LIN {X 0,Y 474.9,Z 291.328,A -85,B 0,C 180,E1 -7380,E2 -7380} C_VEL
LIN {X 0,Y 474.884,Z 291.326,A -85,B 0,C 180,E1 -7382.545,E2 -7382.545} C_VEL
LIN {X 0,Y 474.749,Z 291.35,A -85,B 0,C 180,E1 -7385.948,E2 -7385.948} C_VEL
LIN {X 0,Y 474.718,Z 291.348,A -85,B 0,C 180,E1 -7388.514,E2 -7388.514} C_VEL
LIN {X 0,Y 474.695,Z 291.358,A -85,B 0,C 180,E1 -7391.963,E2 -7391.963} C_VEL
LIN {X 0,Y 474.692,Z 291.354,A -85,B 0,C 180,E1 -7395.777,E2 -7395.777} C_VEL
LIN {X 0,Y 474.655,Z 291.355,A -85,B 0,C 180,E1 -7399.011,E2 -7399.011} C_VEL
LIN {X 0,Y 474.579,Z 291.366,A -85,B 0,C 180,E1 -7401.73,E2 -7401.73} C_VEL
LIN {X 0,Y 474.628,Z 291.364,A -85,B 0,C 180,E1 -7404.495,E2 -7404.495} C_VEL
LIN {X 0,Y 474.665,Z 291.353,A -85,B 0,C 180,E1 -7407.333,E2 -7407.333} C_VEL
LIN {X 0,Y 474.597,Z 291.367,A -85,B 0,C 180,E1 -7410.231,E2 -7410.231} C_VEL
LIN {X 0,Y 474.635,Z 291.358,A -85,B 0,C 180,E1 -7413.221,E2 -7413.221} C_VEL
LIN {X 0,Y 474.581,Z 291.368,A -85,B 0,C 180,E1 -7416.324,E2 -7416.324} C_VEL
LIN {X 0,Y 474.615,Z 291.36,A -85,B 0,C 180,E1 -7419.549,E2 -7419.549} C_VEL
LIN {X 0,Y 474.595,Z 291.369,A -85,B 0,C 180,E1 -7422.937,E2 -7422.937} C_VEL
LIN {X 0,Y 474.597,Z 291.362,A -85,B 0,C 180,E1 -7425.895,E2 -7425.895} C_VEL
LIN {X 0,Y 474.6,Z 291.37,A -85,B 0,C 180,E1 -7429.045,E2 -7429.045} C_VEL
LIN {X 0,Y 474.602,Z 291.362,A -85,B 0,C 180,E1 -7431.706,E2 -7431.706} C_VEL
LIN {X 0,Y 474.617,Z 291.362,A -85,B 0,C 180,E1 -7434.726,E2 -7434.726} C_VEL
LIN {X 0,Y 474.63,Z 291.359,A -85,B 0,C 180,E1 -7437.789,E2 -7437.789} C_VEL
LIN {X 0,Y 474.596,Z 291.365,A -85,B 0,C 180,E1 -7440.891,E2 -7440.891} C_VEL
LIN {X 0,Y 474.578,Z 291.369,A -85,B 0,C 180,E1 -7443.625,E2 -7443.625} C_VEL
LIN {X 0,Y 474.633,Z 291.357,A -85,B 0,C 180,E1 -7446.643,E2 -7446.643} C_VEL
LIN {X 0,Y 474.651,Z 291.357,A -85,B 0,C 180,E1 -7450.09,E2 -7450.09} C_VEL
LIN {X 0,Y 474.643,Z 291.361,A -85,B 0,C 180,E1 -7451.657,E2 -7451.657} C_VEL
LIN {X 0,Y 473.971,Z 291.444,A -85,B 0,C 180,E1 -7452.366,E2 -7452.366} C_VEL
LIN {X 0,Y 471.123,Z 291.802,A -85,B 0,C 180,E1 -7453.518,E2 -7453.518} C_VEL
LIN {X 0,Y 468.714,Z 292.1,A -85,B 0,C 180,E1 -7454.446,E2 -7454.446} C_VEL
LIN {X 0,Y 467.674,Z 292.226,A -85,B 0,C 180,E1 -7455.163,E2 -7455.163} C_VEL
LIN {X 0,Y 467.585,Z 292.237,A -85,B 0,C 180,E1 -7455.406,E2 -7455.406} C_VEL
LIN {X 0,Y 467.636,Z 292.236,A -85,B 0,C 180,E1 -7457.855,E2 -7457.855} C_VEL
LIN {X 0,Y 467.629,Z 292.236,A -85,B 0,C 180,E1 -7461.357,E2 -7461.357} C_VEL
LIN {X 0,Y 467.684,Z 292.306,A -85,B 0,C 180,E1 -7463.313,E2 -7463.313} C_VEL
LIN {X 0,Y 468.568,Z 298.536,A -85,B 0,C 180,E1 -7464.622,E2 -7464.622} C_VEL
LIN {X 0,Y 468.317,Z 310.915,A -85,B 0,C 180,E1 -7467.097,E2 -7467.097} C_VEL
LIN {X 0,Y 471.304,Z 325.673,A -85,B 0,C 180,E1 -7467.437,E2 -7467.437} C_VEL
LIN {X 0,Y 470.534,Z 418.4,A -85,B 0,C 180,E1 -7468.877,E2 -7468.877} C_VEL
LIN {X 0,Y 470.235,Z 431.426,A -85,B 0,C 180,E1 -7469.251,E2 -7469.251} C_VEL
LIN {X 0,Y 469.902,Z 443.958,A -85,B 0,C 180,E1 -7469.786,E2 -7469.786} C_VEL
LIN {X 0,Y 469.513,Z 455.149,A -85,B 0,C 180,E1 -7470.429,E2 -7470.429} C_VEL
LIN {X 0,Y 468.998,Z 466.713,A -85,B 0,C 180,E1 -7471.289,E2 -7471.289} C_VEL
LIN {X 0,Y 468.477,Z 477.124,A -85,B 0,C 180,E1 -7472.257,E2 -7472.257} C_VEL
LIN {X 0,Y 468.064,Z 485.641,A -85,B 0,C 180,E1 -7473.228,E2 -7473.228} C_VEL
LIN {X 0,Y 467.676,Z 493.506,A -85,B 0,C 180,E1 -7474.31,E2 -7474.31} C_VEL
LIN {X 0,Y 467.319,Z 501.212,A -85,B 0,C 180,E1 -7475.61,E2 -7475.61} C_VEL
LIN {X 0,Y 467.128,Z 507.386,A -85,B 0,C 180,E1 -7476.913,E2 -7476.913} C_VEL
LIN {X 0,Y 466.91,Z 512.316,A -85,B 0,C 180,E1 -7478.222,E2 -7478.222} C_VEL
LIN {X 0,Y 466.766,Z 516.123,A -85,B 0,C 180,E1 -7479.534,E2 -7479.534} C_VEL
LIN {X 0,Y 466.713,Z 518.087,A -85,B 0,C 180,E1 -7480.411,E2 -7480.411} C_VEL
LIN {X 0,Y 466.654,Z 520.275,A -85,B 0,C 180,E1 -7481.782,E2 -7481.782} C_VEL
LIN {X 0,Y 466.566,Z 521.392,A -85,B 0,C 180,E1 -7483.059,E2 -7483.059} C_VEL
LIN {X 0,Y 466.536,Z 521.677,A -85,B 0,C 180,E1 -7483.948,E2 -7483.948} C_VEL
LIN {X 0,Y 466.586,Z 521.216,A -85,B 0,C 180,E1 -7485.418,E2 -7485.418} C_VEL
LIN {X 0,Y 466.553,Z 519.949,A -85,B 0,C 180,E1 -7486.632,E2 -7486.632} C_VEL
LIN {X 0,Y 466.652,Z 518.526,A -85,B 0,C 180,E1 -7487.531,E2 -7487.531} C_VEL
LIN {X 0,Y 466.799,Z 515.6,A -85,B 0,C 180,E1 -7488.842,E2 -7488.842} C_VEL
LIN {X 0,Y 466.982,Z 511.277,A -85,B 0,C 180,E1 -7490.252,E2 -7490.252} C_VEL
LIN {X 0,Y 467.214,Z 505.761,A -85,B 0,C 180,E1 -7491.626,E2 -7491.626} C_VEL
LIN {X 0,Y 467.533,Z 498.734,A -85,B 0,C 180,E1 -7493.007,E2 -7493.007} C_VEL
LIN {X 0,Y 467.895,Z 491.468,A -85,B 0,C 180,E1 -7494.162,E2 -7494.162} C_VEL
LIN {X 0,Y 468.379,Z 482.6,A -85,B 0,C 180,E1 -7495.318,E2 -7495.318} C_VEL
LIN {X 0,Y 468.801,Z 473.035,A -85,B 0,C 180,E1 -7496.331,E2 -7496.331} C_VEL
LIN {X 0,Y 469.269,Z 463.203,A -85,B 0,C 180,E1 -7497.18,E2 -7497.18} C_VEL
LIN {X 0,Y 469.812,Z 452.16,A -85,B 0,C 180,E1 -7497.943,E2 -7497.943} C_VEL
LIN {X 0,Y 470.175,Z 440.391,A -85,B 0,C 180,E1 -7498.576,E2 -7498.576} C_VEL
LIN {X 0,Y 470.52,Z 427.541,A -85,B 0,C 180,E1 -7499.072,E2 -7499.072} C_VEL
LIN {X 0,Y 470.719,Z 414.32,A -85,B 0,C 180,E1 -7499.396,E2 -7499.396} C_VEL
LIN {X 0,Y 471.527,Z 325.723,A -85,B 0,C 180,E1 -7500.767,E2 -7500.767} C_VEL
LIN {X 0,Y 468.488,Z 310.771,A -85,B 0,C 180,E1 -7501.149,E2 -7501.149} C_VEL
LIN {X 0,Y 468.731,Z 298.881,A -85,B 0,C 180,E1 -7503.467,E2 -7503.467} C_VEL
LIN {X 0,Y 467.617,Z 292.239,A -85,B 0,C 180,E1 -7504.861,E2 -7504.861} C_VEL
LIN {X 0,Y 467.563,Z 292.243,A -85,B 0,C 180,E1 -7508.591,E2 -7508.591} C_VEL
LIN {X 0,Y 467.579,Z 292.239,A -85,B 0,C 180,E1 -7511.403,E2 -7511.403} C_VEL
LIN {X 0,Y 467.554,Z 292.244,A -85,B 0,C 180,E1 -7513.821,E2 -7513.821} C_VEL
LIN {X 0,Y 467.556,Z 292.245,A -85,B 0,C 180,E1 -7516.255,E2 -7516.255} C_VEL
LIN {X 0,Y 467.58,Z 292.246,A -85,B 0,C 180,E1 -7518.723,E2 -7518.723} C_VEL
LIN {X 0,Y 467.566,Z 292.238,A -85,B 0,C 180,E1 -7521.955,E2 -7521.955} C_VEL
LIN {X 0,Y 467.565,Z 292.244,A -85,B 0,C 180,E1 -7525.167,E2 -7525.167} C_VEL
LIN {X 0,Y 467.583,Z 292.237,A -85,B 0,C 180,E1 -7528.26,E2 -7528.26} C_VEL
LIN {X 0,Y 467.578,Z 292.243,A -85,B 0,C 180,E1 -7531.25,E2 -7531.25} C_VEL
LIN {X 0,Y 467.611,Z 292.232,A -85,B 0,C 180,E1 -7534.16,E2 -7534.16} C_VEL
LIN {X 0,Y 467.577,Z 292.24,A -85,B 0,C 180,E1 -7536.996,E2 -7536.996} C_VEL
LIN {X 0,Y 467.623,Z 292.232,A -85,B 0,C 180,E1 -7539.777,E2 -7539.777} C_VEL
LIN {X 0,Y 467.607,Z 292.232,A -85,B 0,C 180,E1 -7542.507,E2 -7542.507} C_VEL
LIN {X 0,Y 467.606,Z 292.236,A -85,B 0,C 180,E1 -7545.196,E2 -7545.196} C_VEL
LIN {X 0,Y 467.656,Z 292.232,A -85,B 0,C 180,E1 -7547.854,E2 -7547.854} C_VEL
LIN {X 0,Y 467.681,Z 292.222,A -85,B 0,C 180,E1 -7551.357,E2 -7551.357} C_VEL
LIN {X 0,Y 467.734,Z 292.221,A -85,B 0,C 180,E1 -7553.962,E2 -7553.962} C_VEL
LIN {X 0,Y 467.859,Z 292.202,A -85,B 0,C 180,E1 -7557.417,E2 -7557.417} C_VEL
LIN {X 0,Y 467.882,Z 292.2,A -85,B 0,C 180,E1 -7560,E2 -7560} C_VEL
LIN {X 0,Y 467.859,Z 292.202,A -85,B 0,C 180,E1 -7562.583,E2 -7562.583} C_VEL
LIN {X 0,Y 467.734,Z 292.218,A -85,B 0,C 180,E1 -7566.037,E2 -7566.037} C_VEL
LIN {X 0,Y 467.68,Z 292.226,A -85,B 0,C 180,E1 -7568.643,E2 -7568.643} C_VEL
LIN {X 0,Y 467.656,Z 292.226,A -85,B 0,C 180,E1 -7572.145,E2 -7572.145} C_VEL
LIN {X 0,Y 467.639,Z 292.226,A -85,B 0,C 180,E1 -7575.695,E2 -7575.695} C_VEL
LIN {X 0,Y 467.617,Z 292.237,A -85,B 0,C 180,E1 -7578.764,E2 -7578.764} C_VEL
LIN {X 0,Y 467.58,Z 292.234,A -85,B 0,C 180,E1 -7581.268,E2 -7581.268} C_VEL
LIN {X 0,Y 467.571,Z 292.238,A -85,B 0,C 180,E1 -7583.943,E2 -7583.943} C_VEL
LIN {X 0,Y 467.616,Z 292.236,A -85,B 0,C 180,E1 -7586.8,E2 -7586.8} C_VEL
LIN {X 0,Y 467.554,Z 292.235,A -85,B 0,C 180,E1 -7589.738,E2 -7589.738} C_VEL
LIN {X 0,Y 467.579,Z 292.242,A -85,B 0,C 180,E1 -7592.759,E2 -7592.759} C_VEL
LIN {X 0,Y 467.553,Z 292.24,A -85,B 0,C 180,E1 -7595.89,E2 -7595.89} C_VEL
LIN {X 0,Y 467.577,Z 292.245,A -85,B 0,C 180,E1 -7599.145,E2 -7599.145} C_VEL
LIN {X 0,Y 467.588,Z 292.237,A -85,B 0,C 180,E1 -7602.567,E2 -7602.567} C_VEL
LIN {X 0,Y 467.567,Z 292.243,A -85,B 0,C 180,E1 -7605.053,E2 -7605.053} C_VEL
LIN {X 0,Y 467.591,Z 292.243,A -85,B 0,C 180,E1 -7607.44,E2 -7607.44} C_VEL
LIN {X 0,Y 467.562,Z 292.236,A -85,B 0,C 180,E1 -7610.853,E2 -7610.853} C_VEL
LIN {X 0,Y 467.562,Z 292.241,A -85,B 0,C 180,E1 -7614.261,E2 -7614.261} C_VEL
LIN {X 0,Y 467.584,Z 292.237,A -85,B 0,C 180,E1 -7617.321,E2 -7617.321} C_VEL
LIN {X 0,Y 467.572,Z 292.24,A -85,B 0,C 180,E1 -7620.667,E2 -7620.667} C_VEL
LIN {X 0,Y 467.673,Z 292.272,A -85,B 0,C 180,E1 -7623.834,E2 -7623.834} C_VEL
LIN {X 0,Y 469.744,Z 302.888,A -85,B 0,C 180,E1 -7625.873,E2 -7625.873} C_VEL
LIN {X 0,Y 469.91,Z 307.191,A -85,B 0,C 180,E1 -7626.65,E2 -7626.65} C_VEL
LIN {X 0,Y 469.071,Z 325.495,A -85,B 0,C 180,E1 -7629.842,E2 -7629.842} C_VEL
LIN {X 0,Y 468.333,Z 343.342,A -85,B 0,C 180,E1 -7632.905,E2 -7632.905} C_VEL
LIN {X 0,Y 471.301,Z 362.787,A -85,B 0,C 180,E1 -7633.335,E2 -7633.335} C_VEL
LIN {X 0,Y 470.598,Z 452.262,A -85,B 0,C 180,E1 -7634.739,E2 -7634.739} C_VEL
LIN {X 0,Y 470.197,Z 466.109,A -85,B 0,C 180,E1 -7635.141,E2 -7635.141} C_VEL
LIN {X 0,Y 469.77,Z 477.981,A -85,B 0,C 180,E1 -7635.653,E2 -7635.653} C_VEL
LIN {X 0,Y 469.201,Z 490.341,A -85,B 0,C 180,E1 -7636.376,E2 -7636.376} C_VEL
LIN {X 0,Y 468.695,Z 501.658,A -85,B 0,C 180,E1 -7637.233,E2 -7637.233} C_VEL
LIN {X 0,Y 468.238,Z 511.919,A -85,B 0,C 180,E1 -7638.199,E2 -7638.199} C_VEL
LIN {X 0,Y 467.792,Z 520.422,A -85,B 0,C 180,E1 -7639.175,E2 -7639.175} C_VEL
LIN {X 0,Y 467.345,Z 529.647,A -85,B 0,C 180,E1 -7640.478,E2 -7640.478} C_VEL
LIN {X 0,Y 467.066,Z 537.077,A -85,B 0,C 180,E1 -7641.781,E2 -7641.781} C_VEL
LIN {X 0,Y 466.851,Z 543.047,A -85,B 0,C 180,E1 -7643.082,E2 -7643.082} C_VEL
LIN {X 0,Y 466.761,Z 547.769,A -85,B 0,C 180,E1 -7644.383,E2 -7644.383} C_VEL
LIN {X 0,Y 466.647,Z 551.376,A -85,B 0,C 180,E1 -7645.681,E2 -7645.681} C_VEL
LIN {X 0,Y 466.69,Z 553.238,A -85,B 0,C 180,E1 -7646.546,E2 -7646.546} C_VEL
LIN {X 0,Y 466.662,Z 554.634,A -85,B 0,C 180,E1 -7647.41,E2 -7647.41} C_VEL
LIN {X 0,Y 466.619,Z 556.239,A -85,B 0,C 180,E1 -7649.136,E2 -7649.136} C_VEL
LIN {X 0,Y 466.6,Z 556.45,A -85,B 0,C 180,E1 -7649.999,E2 -7649.999} C_VEL
LIN {X 0,Y 466.619,Z 556.23,A -85,B 0,C 180,E1 -7650.862,E2 -7650.862} C_VEL
LIN {X 0,Y 466.661,Z 554.618,A -85,B 0,C 180,E1 -7652.589,E2 -7652.589} C_VEL
LIN {X 0,Y 466.69,Z 553.209,A -85,B 0,C 180,E1 -7653.453,E2 -7653.453} C_VEL
LIN {X 0,Y 466.689,Z 550.252,A -85,B 0,C 180,E1 -7654.75,E2 -7654.75} C_VEL
LIN {X 0,Y 466.749,Z 546.248,A -85,B 0,C 180,E1 -7656.05,E2 -7656.05} C_VEL
LIN {X 0,Y 466.925,Z 540.082,A -85,B 0,C 180,E1 -7657.567,E2 -7657.567} C_VEL
LIN {X 0,Y 467.173,Z 533.351,A -85,B 0,C 180,E1 -7658.87,E2 -7658.87} C_VEL
LIN {X 0,Y 467.506,Z 524.996,A -85,B 0,C 180,E1 -7660.173,E2 -7660.173} C_VEL
LIN {X 0,Y 467.959,Z 516.408,A -85,B 0,C 180,E1 -7661.258,E2 -7661.258} C_VEL
LIN {X 0,Y 468.462,Z 506.244,A -85,B 0,C 180,E1 -7662.302,E2 -7662.302} C_VEL
LIN {X 0,Y 468.894,Z 495.29,A -85,B 0,C 180,E1 -7663.212,E2 -7663.212} C_VEL
LIN {X 0,Y 469.375,Z 483.709,A -85,B 0,C 180,E1 -7663.971,E2 -7663.971} C_VEL
LIN {X 0,Y 469.876,Z 471.688,A -85,B 0,C 180,E1 -7664.563,E2 -7664.563} C_VEL
LIN {X 0,Y 470.216,Z 458.667,A -85,B 0,C 180,E1 -7665.023,E2 -7665.023} C_VEL
LIN {X 0,Y 470.529,Z 446.449,A -85,B 0,C 180,E1 -7665.29,E2 -7665.29} C_VEL
LIN {X 0,Y 471.089,Z 362.504,A -85,B 0,C 180,E1 -7666.577,E2 -7666.577} C_VEL
LIN {X 0,Y 468.243,Z 343.622,A -85,B 0,C 180,E1 -7666.968,E2 -7666.968} C_VEL
LIN {X 0,Y 468.939,Z 326.235,A -85,B 0,C 180,E1 -7669.934,E2 -7669.934} C_VEL
LIN {X 0,Y 469.689,Z 307.742,A -85,B 0,C 180,E1 -7673.127,E2 -7673.127} C_VEL
LIN {X 0,Y 469.59,Z 302.323,A -85,B 0,C 180,E1 -7674.084,E2 -7674.084} C_VEL
LIN {X 0,Y 467.647,Z 292.236,A -85,B 0,C 180,E1 -7675.986,E2 -7675.986} C_VEL
LIN {X 0,Y 467.575,Z 292.241,A -85,B 0,C 180,E1 -7678.749,E2 -7678.749} C_VEL
LIN {X 0,Y 467.58,Z 292.239,A -85,B 0,C 180,E1 -7681.739,E2 -7681.739} C_VEL
LIN {X 0,Y 467.564,Z 292.239,A -85,B 0,C 180,E1 -7684.831,E2 -7684.831} C_VEL
LIN {X 0,Y 467.561,Z 292.243,A -85,B 0,C 180,E1 -7688.043,E2 -7688.043} C_VEL
LIN {X 0,Y 467.573,Z 292.237,A -85,B 0,C 180,E1 -7691.276,E2 -7691.276} C_VEL
LIN {X 0,Y 467.549,Z 292.241,A -85,B 0,C 180,E1 -7693.82,E2 -7693.82} C_VEL
LIN {X 0,Y 467.563,Z 292.243,A -85,B 0,C 180,E1 -7696.256,E2 -7696.256} C_VEL
LIN {X 0,Y 467.576,Z 292.243,A -85,B 0,C 180,E1 -7698.722,E2 -7698.722} C_VEL
LIN {X 0,Y 467.56,Z 292.239,A -85,B 0,C 180,E1 -7701.955,E2 -7701.955} C_VEL
LIN {X 0,Y 467.56,Z 292.241,A -85,B 0,C 180,E1 -7705.167,E2 -7705.167} C_VEL
LIN {X 0,Y 467.58,Z 292.237,A -85,B 0,C 180,E1 -7708.26,E2 -7708.26} C_VEL
LIN {X 0,Y 467.574,Z 292.241,A -85,B 0,C 180,E1 -7711.25,E2 -7711.25} C_VEL
LIN {X 0,Y 467.603,Z 292.233,A -85,B 0,C 180,E1 -7714.16,E2 -7714.16} C_VEL
LIN {X 0,Y 467.568,Z 292.245,A -85,B 0,C 180,E1 -7716.995,E2 -7716.995} C_VEL
LIN {X 0,Y 467.613,Z 292.233,A -85,B 0,C 180,E1 -7719.777,E2 -7719.777} C_VEL
LIN {X 0,Y 467.599,Z 292.234,A -85,B 0,C 180,E1 -7722.506,E2 -7722.506} C_VEL
LIN {X 0,Y 467.6,Z 292.241,A -85,B 0,C 180,E1 -7725.196,E2 -7725.196} C_VEL
LIN {X 0,Y 467.647,Z 292.23,A -85,B 0,C 180,E1 -7727.854,E2 -7727.854} C_VEL
LIN {X 0,Y 467.673,Z 292.232,A -85,B 0,C 180,E1 -7731.357,E2 -7731.357} C_VEL
LIN {X 0,Y 467.733,Z 292.219,A -85,B 0,C 180,E1 -7733.963,E2 -7733.963} C_VEL
LIN {X 0,Y 467.849,Z 292.208,A -85,B 0,C 180,E1 -7737.417,E2 -7737.417} C_VEL
LIN {X 0,Y 467.871,Z 292.204,A -85,B 0,C 180,E1 -7740,E2 -7740} C_VEL
LIN {X 0,Y 467.85,Z 292.202,A -85,B 0,C 180,E1 -7742.583,E2 -7742.583} C_VEL
LIN {X 0,Y 467.712,Z 292.225,A -85,B 0,C 180,E1 -7746.038,E2 -7746.038} C_VEL
LIN {X 0,Y 467.671,Z 292.225,A -85,B 0,C 180,E1 -7748.643,E2 -7748.643} C_VEL
LIN {X 0,Y 467.646,Z 292.234,A -85,B 0,C 180,E1 -7752.146,E2 -7752.146} C_VEL
LIN {X 0,Y 467.657,Z 292.232,A -85,B 0,C 180,E1 -7755.893,E2 -7755.893} C_VEL
LIN {X 0,Y 467.614,Z 292.232,A -85,B 0,C 180,E1 -7759.308,E2 -7759.308} C_VEL
LIN {X 0,Y 467.525,Z 292.249,A -85,B 0,C 180,E1 -7762.074,E2 -7762.074} C_VEL
LIN {X 0,Y 467.574,Z 292.238,A -85,B 0,C 180,E1 -7764.889,E2 -7764.889} C_VEL
LIN {X 0,Y 467.606,Z 292.234,A -85,B 0,C 180,E1 -7767.77,E2 -7767.77} C_VEL
LIN {X 0,Y 467.56,Z 292.24,A -85,B 0,C 180,E1 -7771.046,E2 -7771.046} C_VEL
LIN {X 0,Y 467.581,Z 292.24,A -85,B 0,C 180,E1 -7774.243,E2 -7774.243} C_VEL
LIN {X 0,Y 467.54,Z 292.243,A -85,B 0,C 180,E1 -7777.187,E2 -7777.187} C_VEL
LIN {X 0,Y 467.552,Z 292.242,A -85,B 0,C 180,E1 -7780.267,E2 -7780.267} C_VEL
LIN {X 0,Y 467.554,Z 292.244,A -85,B 0,C 180,E1 -7782.564,E2 -7782.564} C_VEL
LIN {X 0,Y 467.56,Z 292.245,A -85,B 0,C 180,E1 -7785.053,E2 -7785.053} C_VEL
LIN {X 0,Y 467.56,Z 292.244,A -85,B 0,C 180,E1 -7788.726,E2 -7788.726} C_VEL
LIN {X 0,Y 467.557,Z 292.239,A -85,B 0,C 180,E1 -7791.956,E2 -7791.956} C_VEL
LIN {X 0,Y 467.554,Z 292.248,A -85,B 0,C 180,E1 -7795.168,E2 -7795.168} C_VEL
LIN {X 0,Y 467.577,Z 292.236,A -85,B 0,C 180,E1 -7798.261,E2 -7798.261} C_VEL
LIN {X 0,Y 467.542,Z 292.249,A -85,B 0,C 180,E1 -7801.249,E2 -7801.249} C_VEL
LIN {X 0,Y 467.574,Z 292.236,A -85,B 0,C 180,E1 -7804.402,E2 -7804.402} C_VEL
LIN {X 0,Y 467.572,Z 292.24,A -85,B 0,C 180,E1 -7806.997,E2 -7806.997} C_VEL
LIN {X 0,Y 467.621,Z 292.236,A -85,B 0,C 180,E1 -7809.778,E2 -7809.778} C_VEL
LIN {X 0,Y 467.589,Z 292.235,A -85,B 0,C 180,E1 -7812.507,E2 -7812.507} C_VEL
LIN {X 0,Y 467.595,Z 292.236,A -85,B 0,C 180,E1 -7815.197,E2 -7815.197} C_VEL
LIN {X 0,Y 467.585,Z 292.237,A -85,B 0,C 180,E1 -7815.406,E2 -7815.406} C_VEL
LIN {X 0,Y 466.911,Z 292.323,A -85,B 0,C 180,E1 -7816.126,E2 -7816.126} C_VEL
LIN {X 0,Y 464.061,Z 292.677,A -85,B 0,C 180,E1 -7817.294,E2 -7817.294} C_VEL
LIN {X 0,Y 461.656,Z 292.976,A -85,B 0,C 180,E1 -7818.236,E2 -7818.236} C_VEL
LIN {X 0,Y 460.624,Z 293.103,A -85,B 0,C 180,E1 -7818.964,E2 -7818.964} C_VEL
LIN {X 0,Y 460.54,Z 293.114,A -85,B 0,C 180,E1 -7819.21,E2 -7819.21} C_VEL
LIN {X 0,Y 460.664,Z 293.105,A -85,B 0,C 180,E1 -7822.595,E2 -7822.595} C_VEL
LIN {X 0,Y 460.609,Z 293.145,A -85,B 0,C 180,E1 -7823.155,E2 -7823.155} C_VEL
LIN {X 0,Y 461.592,Z 299.679,A -85,B 0,C 180,E1 -7824.54,E2 -7824.54} C_VEL
LIN {X 0,Y 461.36,Z 311.156,A -85,B 0,C 180,E1 -7826.863,E2 -7826.863} C_VEL
LIN {X 0,Y 464.459,Z 327.1,A -85,B 0,C 180,E1 -7827.226,E2 -7827.226} C_VEL
LIN {X 0,Y 463.652,Z 418.705,A -85,B 0,C 180,E1 -7828.671,E2 -7828.671} C_VEL
LIN {X 0,Y 463.342,Z 431.715,A -85,B 0,C 180,E1 -7829.05,E2 -7829.05} C_VEL
LIN {X 0,Y 462.991,Z 444.779,A -85,B 0,C 180,E1 -7829.62,E2 -7829.62} C_VEL
LIN {X 0,Y 462.524,Z 456.608,A -85,B 0,C 180,E1 -7830.327,E2 -7830.327} C_VEL
LIN {X 0,Y 462.003,Z 467.956,A -85,B 0,C 180,E1 -7831.199,E2 -7831.199} C_VEL
LIN {X 0,Y 461.459,Z 478.211,A -85,B 0,C 180,E1 -7832.183,E2 -7832.183} C_VEL
LIN {X 0,Y 460.967,Z 487.43,A -85,B 0,C 180,E1 -7833.278,E2 -7833.278} C_VEL
LIN {X 0,Y 460.554,Z 496.369,A -85,B 0,C 180,E1 -7834.596,E2 -7834.596} C_VEL
LIN {X 0,Y 460.201,Z 503.594,A -85,B 0,C 180,E1 -7835.917,E2 -7835.917} C_VEL
LIN {X 0,Y 460.022,Z 508.475,A -85,B 0,C 180,E1 -7837.021,E2 -7837.021} C_VEL
LIN {X 0,Y 459.828,Z 513.231,A -85,B 0,C 180,E1 -7838.349,E2 -7838.349} C_VEL
LIN {X 0,Y 459.66,Z 516.88,A -85,B 0,C 180,E1 -7839.683,E2 -7839.683} C_VEL
LIN {X 0,Y 459.631,Z 518.758,A -85,B 0,C 180,E1 -7840.573,E2 -7840.573} C_VEL
LIN {X 0,Y 459.574,Z 520.641,A -85,B 0,C 180,E1 -7841.841,E2 -7841.841} C_VEL
LIN {X 0,Y 459.473,Z 521.77,A -85,B 0,C 180,E1 -7843.264,E2 -7843.264} C_VEL
LIN {X 0,Y 459.455,Z 521.949,A -85,B 0,C 180,E1 -7844.167,E2 -7844.167} C_VEL
LIN {X 0,Y 459.497,Z 521.443,A -85,B 0,C 180,E1 -7845.509,E2 -7845.509} C_VEL
LIN {X 0,Y 459.507,Z 519.945,A -85,B 0,C 180,E1 -7846.894,E2 -7846.894} C_VEL
LIN {X 0,Y 459.711,Z 516.696,A -85,B 0,C 180,E1 -7848.585,E2 -7848.585} C_VEL
LIN {X 0,Y 459.903,Z 512.386,A -85,B 0,C 180,E1 -7850.111,E2 -7850.111} C_VEL
LIN {X 0,Y 460.13,Z 507.155,A -85,B 0,C 180,E1 -7851.505,E2 -7851.505} C_VEL
LIN {X 0,Y 460.446,Z 500.43,A -85,B 0,C 180,E1 -7852.906,E2 -7852.906} C_VEL
LIN {X 0,Y 460.906,Z 491.907,A -85,B 0,C 180,E1 -7854.312,E2 -7854.312} C_VEL
LIN {X 0,Y 461.434,Z 483.171,A -85,B 0,C 180,E1 -7855.474,E2 -7855.474} C_VEL
LIN {X 0,Y 461.897,Z 473.204,A -85,B 0,C 180,E1 -7856.549,E2 -7856.549} C_VEL
LIN {X 0,Y 462.548,Z 462.326,A -85,B 0,C 180,E1 -7857.486,E2 -7857.486} C_VEL
LIN {X 0,Y 463.034,Z 450.973,A -85,B 0,C 180,E1 -7858.265,E2 -7858.265} C_VEL
LIN {X 0,Y 463.415,Z 439.485,A -85,B 0,C 180,E1 -7858.871,E2 -7858.871} C_VEL
LIN {X 0,Y 463.732,Z 426.718,A -85,B 0,C 180,E1 -7859.353,E2 -7859.353} C_VEL
LIN {X 0,Y 463.93,Z 414.423,A -85,B 0,C 180,E1 -7859.65,E2 -7859.65} C_VEL
LIN {X 0,Y 464.743,Z 326.423,A -85,B 0,C 180,E1 -7861.035,E2 -7861.035} C_VEL
LIN {X 0,Y 461.62,Z 311.018,A -85,B 0,C 180,E1 -7861.441,E2 -7861.441} C_VEL
LIN {X 0,Y 461.79,Z 299.36,A -85,B 0,C 180,E1 -7863.745,E2 -7863.745} C_VEL
LIN {X 0,Y 460.554,Z 293.118,A -85,B 0,C 180,E1 -7865.091,E2 -7865.091} C_VEL
LIN {X 0,Y 460.537,Z 293.117,A -85,B 0,C 180,E1 -7868.896,E2 -7868.896} C_VEL
LIN {X 0,Y 460.525,Z 293.122,A -85,B 0,C 180,E1 -7872.181,E2 -7872.181} C_VEL
LIN {X 0,Y 460.516,Z 293.12,A -85,B 0,C 180,E1 -7875.411,E2 -7875.411} C_VEL
LIN {X 0,Y 460.534,Z 293.122,A -85,B 0,C 180,E1 -7878.397,E2 -7878.397} C_VEL
LIN {X 0,Y 460.527,Z 293.117,A -85,B 0,C 180,E1 -7881.267,E2 -7881.267} C_VEL
LIN {X 0,Y 460.511,Z 293.122,A -85,B 0,C 180,E1 -7884.554,E2 -7884.554} C_VEL
LIN {X 0,Y 460.532,Z 293.115,A -85,B 0,C 180,E1 -7887.715,E2 -7887.715} C_VEL
LIN {X 0,Y 460.541,Z 293.116,A -85,B 0,C 180,E1 -7890.769,E2 -7890.769} C_VEL
LIN {X 0,Y 460.564,Z 293.111,A -85,B 0,C 180,E1 -7893.735,E2 -7893.735} C_VEL
LIN {X 0,Y 460.546,Z 293.113,A -85,B 0,C 180,E1 -7896.624,E2 -7896.624} C_VEL
LIN {X 0,Y 460.552,Z 293.117,A -85,B 0,C 180,E1 -7899.453,E2 -7899.453} C_VEL
LIN {X 0,Y 460.557,Z 293.11,A -85,B 0,C 180,E1 -7902.23,E2 -7902.23} C_VEL
LIN {X 0,Y 460.565,Z 293.111,A -85,B 0,C 180,E1 -7904.965,E2 -7904.965} C_VEL
LIN {X 0,Y 460.611,Z 293.105,A -85,B 0,C 180,E1 -7908.559,E2 -7908.559} C_VEL
LIN {X 0,Y 460.695,Z 293.098,A -85,B 0,C 180,E1 -7912.108,E2 -7912.108} C_VEL
LIN {X 0,Y 460.693,Z 293.092,A -85,B 0,C 180,E1 -7914.748,E2 -7914.748} C_VEL
LIN {X 0,Y 460.799,Z 293.081,A -85,B 0,C 180,E1 -7917.377,E2 -7917.377} C_VEL
LIN {X 0,Y 460.852,Z 293.075,A -85,B 0,C 180,E1 -7920,E2 -7920} C_VEL
LIN {X 0,Y 460.8,Z 293.082,A -85,B 0,C 180,E1 -7922.622,E2 -7922.622} C_VEL
LIN {X 0,Y 460.7,Z 293.093,A -85,B 0,C 180,E1 -7926.13,E2 -7926.13} C_VEL
LIN {X 0,Y 460.627,Z 293.103,A -85,B 0,C 180,E1 -7928.776,E2 -7928.776} C_VEL
LIN {X 0,Y 460.613,Z 293.108,A -85,B 0,C 180,E1 -7932.445,E2 -7932.445} C_VEL
LIN {X 0,Y 460.6,Z 293.105,A -85,B 0,C 180,E1 -7935.998,E2 -7935.998} C_VEL
LIN {X 0,Y 460.571,Z 293.113,A -85,B 0,C 180,E1 -7938.902,E2 -7938.902} C_VEL
LIN {X 0,Y 460.516,Z 293.113,A -85,B 0,C 180,E1 -7941.486,E2 -7941.486} C_VEL
LIN {X 0,Y 460.538,Z 293.117,A -85,B 0,C 180,E1 -7944.333,E2 -7944.333} C_VEL
LIN {X 0,Y 460.573,Z 293.113,A -85,B 0,C 180,E1 -7947.244,E2 -7947.244} C_VEL
LIN {X 0,Y 460.511,Z 293.113,A -85,B 0,C 180,E1 -7950.24,E2 -7950.24} C_VEL
LIN {X 0,Y 460.52,Z 293.117,A -85,B 0,C 180,E1 -7953.326,E2 -7953.326} C_VEL
LIN {X 0,Y 460.477,Z 293.123,A -85,B 0,C 180,E1 -7956.53,E2 -7956.53} C_VEL
LIN {X 0,Y 460.528,Z 293.115,A -85,B 0,C 180,E1 -7959.863,E2 -7959.863} C_VEL
LIN {X 0,Y 460.514,Z 293.121,A -85,B 0,C 180,E1 -7962.9,E2 -7962.9} C_VEL
LIN {X 0,Y 460.51,Z 293.121,A -85,B 0,C 180,E1 -7965.831,E2 -7965.831} C_VEL
LIN {X 0,Y 460.532,Z 293.117,A -85,B 0,C 180,E1 -7968.989,E2 -7968.989} C_VEL
LIN {X 0,Y 460.52,Z 293.116,A -85,B 0,C 180,E1 -7971.266,E2 -7971.266} C_VEL
LIN {X 0,Y 460.512,Z 293.118,A -85,B 0,C 180,E1 -7974.554,E2 -7974.554} C_VEL
LIN {X 0,Y 460.534,Z 293.12,A -85,B 0,C 180,E1 -7977.716,E2 -7977.716} C_VEL
LIN {X 0,Y 460.542,Z 293.116,A -85,B 0,C 180,E1 -7980.769,E2 -7980.769} C_VEL
LIN {X 0,Y 460.61,Z 293.179,A -85,B 0,C 180,E1 -7983.585,E2 -7983.585} C_VEL
LIN {X 0,Y 462.851,Z 304.474,A -85,B 0,C 180,E1 -7985.797,E2 -7985.797} C_VEL
LIN {X 0,Y 462.931,Z 309.699,A -85,B 0,C 180,E1 -7986.751,E2 -7986.751} C_VEL
LIN {X 0,Y 462.115,Z 326.694,A -85,B 0,C 180,E1 -7989.757,E2 -7989.757} C_VEL
LIN {X 0,Y 461.366,Z 343.006,A -85,B 0,C 180,E1 -7992.604,E2 -7992.604} C_VEL
LIN {X 0,Y 464.549,Z 364.085,A -85,B 0,C 180,E1 -7993.088,E2 -7993.088} C_VEL
LIN {X 0,Y 463.805,Z 451.723,A -85,B 0,C 180,E1 -7994.481,E2 -7994.481} C_VEL
LIN {X 0,Y 463.425,Z 464.897,A -85,B 0,C 180,E1 -7994.863,E2 -7994.863} C_VEL
LIN {X 0,Y 462.917,Z 477.013,A -85,B 0,C 180,E1 -7995.38,E2 -7995.38} C_VEL
LIN {X 0,Y 462.419,Z 488.45,A -85,B 0,C 180,E1 -7996.038,E2 -7996.038} C_VEL
LIN {X 0,Y 461.827,Z 500.542,A -85,B 0,C 180,E1 -7996.945,E2 -7996.945} C_VEL
LIN {X 0,Y 461.279,Z 511.832,A -85,B 0,C 180,E1 -7998.018,E2 -7998.018} C_VEL
LIN {X 0,Y 460.797,Z 520.291,A -85,B 0,C 180,E1 -7999.009,E2 -7999.009} C_VEL
LIN {X 0,Y 460.331,Z 529.474,A -85,B 0,C 180,E1 -8000.331,E2 -8000.331} C_VEL
LIN {X 0,Y 460.002,Z 536.878,A -85,B 0,C 180,E1 -8001.654,E2 -8001.654} C_VEL
LIN {X 0,Y 459.769,Z 542.833,A -85,B 0,C 180,E1 -8002.975,E2 -8002.975} C_VEL
LIN {X 0,Y 459.657,Z 547.544,A -85,B 0,C 180,E1 -8004.296,E2 -8004.296} C_VEL
LIN {X 0,Y 459.565,Z 551.141,A -85,B 0,C 180,E1 -8005.614,E2 -8005.614} C_VEL
LIN {X 0,Y 459.585,Z 552.995,A -85,B 0,C 180,E1 -8006.493,E2 -8006.493} C_VEL
LIN {X 0,Y 459.584,Z 554.385,A -85,B 0,C 180,E1 -8007.37,E2 -8007.37} C_VEL
LIN {X 0,Y 459.523,Z 555.981,A -85,B 0,C 180,E1 -8009.123,E2 -8009.123} C_VEL
LIN {X 0,Y 459.532,Z 556.186,A -85,B 0,C 180,E1 -8009.999,E2 -8009.999} C_VEL
LIN {X 0,Y 459.552,Z 555.959,A -85,B 0,C 180,E1 -8010.876,E2 -8010.876} C_VEL
LIN {X 0,Y 459.584,Z 554.336,A -85,B 0,C 180,E1 -8012.629,E2 -8012.629} C_VEL
LIN {X 0,Y 459.586,Z 552.918,A -85,B 0,C 180,E1 -8013.506,E2 -8013.506} C_VEL
LIN {X 0,Y 459.616,Z 549.953,A -85,B 0,C 180,E1 -8014.824,E2 -8014.824} C_VEL
LIN {X 0,Y 459.713,Z 544.889,A -85,B 0,C 180,E1 -8016.43,E2 -8016.43} C_VEL
LIN {X 0,Y 459.891,Z 538.737,A -85,B 0,C 180,E1 -8017.905,E2 -8017.905} C_VEL
LIN {X 0,Y 460.186,Z 531.761,A -85,B 0,C 180,E1 -8019.227,E2 -8019.227} C_VEL
LIN {X 0,Y 460.57,Z 523.009,A -85,B 0,C 180,E1 -8020.55,E2 -8020.55} C_VEL
LIN {X 0,Y 461.057,Z 514.037,A -85,B 0,C 180,E1 -8021.652,E2 -8021.652} C_VEL
LIN {X 0,Y 461.594,Z 503.056,A -85,B 0,C 180,E1 -8022.745,E2 -8022.745} C_VEL
LIN {X 0,Y 462.096,Z 491.713,A -85,B 0,C 180,E1 -8023.634,E2 -8023.634} C_VEL
LIN {X 0,Y 462.626,Z 479.098,A -85,B 0,C 180,E1 -8024.403,E2 -8024.403} C_VEL
LIN {X 0,Y 463.112,Z 466.125,A -85,B 0,C 180,E1 -8024.978,E2 -8024.978} C_VEL
LIN {X 0,Y 463.527,Z 453.373,A -85,B 0,C 180,E1 -8025.358,E2 -8025.358} C_VEL
LIN {X 0,Y 463.816,Z 422.492,A -85,B 0,C 180,E1 -8025.869,E2 -8025.869} C_VEL
LIN {X 0,Y 464.104,Z 362.333,A -85,B 0,C 180,E1 -8026.809,E2 -8026.809} C_VEL
LIN {X 0,Y 461.257,Z 343.237,A -85,B 0,C 180,E1 -8027.231,E2 -8027.231} C_VEL
LIN {X 0,Y 461.93,Z 327.143,A -85,B 0,C 180,E1 -8030.018,E2 -8030.018} C_VEL
LIN {X 0,Y 462.743,Z 308.632,A -85,B 0,C 180,E1 -8033.257,E2 -8033.257} C_VEL
LIN {X 0,Y 462.779,Z 304.647,A -85,B 0,C 180,E1 -8033.968,E2 -8033.968} C_VEL
LIN {X 0,Y 460.61,Z 293.112,A -85,B 0,C 180,E1 -8036.168,E2 -8036.168} C_VEL
LIN {X 0,Y 460.538,Z 293.117,A -85,B 0,C 180,E1 -8039.23,E2 -8039.23} C_VEL
LIN {X 0,Y 460.529,Z 293.121,A -85,B 0,C 180,E1 -8042.283,E2 -8042.283} C_VEL
LIN {X 0,Y 460.509,Z 293.117,A -85,B 0,C 180,E1 -8045.444,E2 -8045.444} C_VEL
LIN {X 0,Y 460.53,Z 293.116,A -85,B 0,C 180,E1 -8048.895,E2 -8048.895} C_VEL
LIN {X 0,Y 460.518,Z 293.121,A -85,B 0,C 180,E1 -8052.18,E2 -8052.18} C_VEL
LIN {X 0,Y 460.515,Z 293.116,A -85,B 0,C 180,E1 -8055.411,E2 -8055.411} C_VEL
LIN {X 0,Y 460.529,Z 293.12,A -85,B 0,C 180,E1 -8058.396,E2 -8058.396} C_VEL
LIN {X 0,Y 460.52,Z 293.117,A -85,B 0,C 180,E1 -8061.266,E2 -8061.266} C_VEL
LIN {X 0,Y 460.506,Z 293.123,A -85,B 0,C 180,E1 -8064.554,E2 -8064.554} C_VEL
LIN {X 0,Y 460.526,Z 293.115,A -85,B 0,C 180,E1 -8067.715,E2 -8067.715} C_VEL
LIN {X 0,Y 460.539,Z 293.12,A -85,B 0,C 180,E1 -8070.769,E2 -8070.769} C_VEL
LIN {X 0,Y 460.56,Z 293.111,A -85,B 0,C 180,E1 -8073.734,E2 -8073.734} C_VEL
LIN {X 0,Y 460.537,Z 293.116,A -85,B 0,C 180,E1 -8076.623,E2 -8076.623} C_VEL
LIN {X 0,Y 460.542,Z 293.117,A -85,B 0,C 180,E1 -8079.452,E2 -8079.452} C_VEL
LIN {X 0,Y 460.549,Z 293.112,A -85,B 0,C 180,E1 -8082.23,E2 -8082.23} C_VEL
LIN {X 0,Y 460.558,Z 293.115,A -85,B 0,C 180,E1 -8084.965,E2 -8084.965} C_VEL
LIN {X 0,Y 460.604,Z 293.105,A -85,B 0,C 180,E1 -8088.559,E2 -8088.559} C_VEL
LIN {X 0,Y 460.685,Z 293.096,A -85,B 0,C 180,E1 -8092.108,E2 -8092.108} C_VEL
LIN {X 0,Y 460.687,Z 293.095,A -85,B 0,C 180,E1 -8094.748,E2 -8094.748} C_VEL
LIN {X 0,Y 460.814,Z 293.084,A -85,B 0,C 180,E1 -8097.378,E2 -8097.378} C_VEL
LIN {X 0,Y 460.842,Z 293.079,A -85,B 0,C 180,E1 -8100,E2 -8100} C_VEL
LIN {X 0,Y 460.815,Z 293.079,A -85,B 0,C 180,E1 -8102.622,E2 -8102.622} C_VEL
LIN {X 0,Y 460.676,Z 293.1,A -85,B 0,C 180,E1 -8106.13,E2 -8106.13} C_VEL
LIN {X 0,Y 460.619,Z 293.103,A -85,B 0,C 180,E1 -8108.776,E2 -8108.776} C_VEL
LIN {X 0,Y 460.604,Z 293.108,A -85,B 0,C 180,E1 -8112.445,E2 -8112.445} C_VEL
LIN {X 0,Y 460.613,Z 293.111,A -85,B 0,C 180,E1 -8116.008,E2 -8116.008} C_VEL
LIN {X 0,Y 460.559,Z 293.112,A -85,B 0,C 180,E1 -8119.616,E2 -8119.616} C_VEL
LIN {X 0,Y 460.501,Z 293.124,A -85,B 0,C 180,E1 -8122.429,E2 -8122.429} C_VEL
LIN {X 0,Y 460.538,Z 293.115,A -85,B 0,C 180,E1 -8125.797,E2 -8125.797} C_VEL
LIN {X 0,Y 460.54,Z 293.119,A -85,B 0,C 180,E1 -8128.234,E2 -8128.234} C_VEL
LIN {X 0,Y 460.513,Z 293.117,A -85,B 0,C 180,E1 -8131.284,E2 -8131.284} C_VEL
LIN {X 0,Y 460.524,Z 293.122,A -85,B 0,C 180,E1 -8134.506,E2 -8134.506} C_VEL
LIN {X 0,Y 460.493,Z 293.119,A -85,B 0,C 180,E1 -8137.624,E2 -8137.624} C_VEL
LIN {X 0,Y 460.513,Z 293.121,A -85,B 0,C 180,E1 -8141.014,E2 -8141.014} C_VEL
LIN {X 0,Y 460.499,Z 293.119,A -85,B 0,C 180,E1 -8144.17,E2 -8144.17} C_VEL
LIN {X 0,Y 460.475,Z 293.127,A -85,B 0,C 180,E1 -8147.105,E2 -8147.105} C_VEL
LIN {X 0,Y 460.508,Z 293.117,A -85,B 0,C 180,E1 -8150.137,E2 -8150.137} C_VEL
LIN {X 0,Y 460.469,Z 293.125,A -85,B 0,C 180,E1 -8153.471,E2 -8153.471} C_VEL
LIN {X 0,Y 460.516,Z 293.118,A -85,B 0,C 180,E1 -8156.675,E2 -8156.675} C_VEL
LIN {X 0,Y 460.5,Z 293.12,A -85,B 0,C 180,E1 -8159.76,E2 -8159.76} C_VEL
LIN {X 0,Y 460.486,Z 293.121,A -85,B 0,C 180,E1 -8162.752,E2 -8162.752} C_VEL
LIN {X 0,Y 460.514,Z 293.121,A -85,B 0,C 180,E1 -8165.667,E2 -8165.667} C_VEL
LIN {X 0,Y 460.521,Z 293.115,A -85,B 0,C 180,E1 -8168.579,E2 -8168.579} C_VEL
LIN {X 0,Y 460.584,Z 293.112,A -85,B 0,C 180,E1 -8171.312,E2 -8171.312} C_VEL
LIN {X 0,Y 460.605,Z 293.108,A -85,B 0,C 180,E1 -8174.06,E2 -8174.06} C_VEL
LIN {X 0,Y 460.602,Z 293.113,A -85,B 0,C 180,E1 -8177.666,E2 -8177.666} C_VEL
LIN {X 0,Y 460.54,Z 293.114,A -85,B 0,C 180,E1 -8179.21,E2 -8179.21} C_VEL
LIN {X 0,Y 459.864,Z 293.205,A -85,B 0,C 180,E1 -8179.697,E2 -8179.697} C_VEL
LIN {X 0,Y 457.034,Z 293.555,A -85,B 0,C 180,E1 -8180.459,E2 -8180.459} C_VEL
LIN {X 0,Y 454.207,Z 293.907,A -85,B 0,C 180,E1 -8181.23,E2 -8181.23} C_VEL
LIN {X 0,Y 453.555,Z 293.99,A -85,B 0,C 180,E1 -8181.727,E2 -8181.727} C_VEL
LIN {X 0,Y 453.57,Z 293.995,A -85,B 0,C 180,E1 -8182.992,E2 -8182.992} C_VEL
LIN {X 0,Y 454.638,Z 300.807,A -85,B 0,C 180,E1 -8184.456,E2 -8184.456} C_VEL
LIN {X 0,Y 454.402,Z 311.37,A -85,B 0,C 180,E1 -8186.616,E2 -8186.616} C_VEL
LIN {X 0,Y 457.623,Z 327.669,A -85,B 0,C 180,E1 -8186.996,E2 -8186.996} C_VEL
LIN {X 0,Y 456.777,Z 419.008,A -85,B 0,C 180,E1 -8188.458,E2 -8188.458} C_VEL
LIN {X 0,Y 456.462,Z 431.998,A -85,B 0,C 180,E1 -8188.843,E2 -8188.843} C_VEL
LIN {X 0,Y 456.107,Z 444.51,A -85,B 0,C 180,E1 -8189.394,E2 -8189.394} C_VEL
LIN {X 0,Y 455.637,Z 456.482,A -85,B 0,C 180,E1 -8190.111,E2 -8190.111} C_VEL
LIN {X 0,Y 455.07,Z 467.909,A -85,B 0,C 180,E1 -8190.996,E2 -8190.996} C_VEL
LIN {X 0,Y 454.483,Z 478.223,A -85,B 0,C 180,E1 -8191.995,E2 -8191.995} C_VEL
LIN {X 0,Y 454,Z 487.493,A -85,B 0,C 180,E1 -8193.106,E2 -8193.106} C_VEL
LIN {X 0,Y 453.534,Z 496.47,A -85,B 0,C 180,E1 -8194.444,E2 -8194.444} C_VEL
LIN {X 0,Y 453.141,Z 503.727,A -85,B 0,C 180,E1 -8195.786,E2 -8195.786} C_VEL
LIN {X 0,Y 452.941,Z 509.532,A -85,B 0,C 180,E1 -8197.131,E2 -8197.131} C_VEL
LIN {X 0,Y 452.729,Z 514.119,A -85,B 0,C 180,E1 -8198.481,E2 -8198.481} C_VEL
LIN {X 0,Y 452.558,Z 517.614,A -85,B 0,C 180,E1 -8199.836,E2 -8199.836} C_VEL
LIN {X 0,Y 452.536,Z 519.352,A -85,B 0,C 180,E1 -8200.741,E2 -8200.741} C_VEL
LIN {X 0,Y 452.473,Z 520.983,A -85,B 0,C 180,E1 -8201.89,E2 -8201.89} C_VEL
LIN {X 0,Y 452.377,Z 522.112,A -85,B 0,C 180,E1 -8203.476,E2 -8203.476} C_VEL
LIN {X 0,Y 452.362,Z 522.179,A -85,B 0,C 180,E1 -8204.394,E2 -8204.394} C_VEL
LIN {X 0,Y 452.421,Z 521.665,A -85,B 0,C 180,E1 -8205.608,E2 -8205.608} C_VEL
LIN {X 0,Y 452.435,Z 519.887,A -85,B 0,C 180,E1 -8207.166,E2 -8207.166} C_VEL
LIN {X 0,Y 452.638,Z 516.88,A -85,B 0,C 180,E1 -8208.713,E2 -8208.713} C_VEL
LIN {X 0,Y 452.815,Z 513.478,A -85,B 0,C 180,E1 -8209.966,E2 -8209.966} C_VEL
LIN {X 0,Y 453.061,Z 508.198,A -85,B 0,C 180,E1 -8211.449,E2 -8211.449} C_VEL
LIN {X 0,Y 453.362,Z 502.06,A -85,B 0,C 180,E1 -8212.802,E2 -8212.802} C_VEL
LIN {X 0,Y 453.797,Z 495.057,A -85,B 0,C 180,E1 -8214.049,E2 -8214.049} C_VEL
LIN {X 0,Y 454.236,Z 487.313,A -85,B 0,C 180,E1 -8215.182,E2 -8215.182} C_VEL
LIN {X 0,Y 454.824,Z 476.918,A -85,B 0,C 180,E1 -8216.411,E2 -8216.411} C_VEL
LIN {X 0,Y 455.446,Z 465.915,A -85,B 0,C 180,E1 -8217.452,E2 -8217.452} C_VEL
LIN {X 0,Y 456.068,Z 454.713,A -85,B 0,C 180,E1 -8218.285,E2 -8218.285} C_VEL
LIN {X 0,Y 456.509,Z 442.108,A -85,B 0,C 180,E1 -8219.009,E2 -8219.009} C_VEL
LIN {X 0,Y 456.882,Z 429.879,A -85,B 0,C 180,E1 -8219.52,E2 -8219.52} C_VEL
LIN {X 0,Y 457.2,Z 416.548,A -85,B 0,C 180,E1 -8219.877,E2 -8219.877} C_VEL
LIN {X 0,Y 458.087,Z 327.531,A -85,B 0,C 180,E1 -8221.305,E2 -8221.305} C_VEL
LIN {X 0,Y 454.714,Z 311.314,A -85,B 0,C 180,E1 -8221.734,E2 -8221.734} C_VEL
LIN {X 0,Y 454.884,Z 301.023,A -85,B 0,C 180,E1 -8223.794,E2 -8223.794} C_VEL
LIN {X 0,Y 453.491,Z 293.998,A -85,B 0,C 180,E1 -8225.328,E2 -8225.328} C_VEL
LIN {X 0,Y 453.463,Z 294.001,A -85,B 0,C 180,E1 -8228.312,E2 -8228.312} C_VEL
LIN {X 0,Y 453.496,Z 293.998,A -85,B 0,C 180,E1 -8230.609,E2 -8230.609} C_VEL
LIN {X 0,Y 453.457,Z 294,A -85,B 0,C 180,E1 -8233.244,E2 -8233.244} C_VEL
LIN {X 0,Y 453.465,Z 293.999,A -85,B 0,C 180,E1 -8235.779,E2 -8235.779} C_VEL
LIN {X 0,Y 453.481,Z 293.999,A -85,B 0,C 180,E1 -8238.209,E2 -8238.209} C_VEL
LIN {X 0,Y 453.517,Z 293.989,A -85,B 0,C 180,E1 -8240.79,E2 -8240.79} C_VEL
LIN {X 0,Y 453.455,Z 293.997,A -85,B 0,C 180,E1 -8243.917,E2 -8243.917} C_VEL
LIN {X 0,Y 453.484,Z 293.998,A -85,B 0,C 180,E1 -8247.151,E2 -8247.151} C_VEL
LIN {X 0,Y 453.476,Z 293.991,A -85,B 0,C 180,E1 -8250.268,E2 -8250.268} C_VEL
LIN {X 0,Y 453.508,Z 293.993,A -85,B 0,C 180,E1 -8253.294,E2 -8253.294} C_VEL
LIN {X 0,Y 453.503,Z 293.989,A -85,B 0,C 180,E1 -8256.239,E2 -8256.239} C_VEL
LIN {X 0,Y 453.483,Z 293.998,A -85,B 0,C 180,E1 -8259.118,E2 -8259.118} C_VEL
LIN {X 0,Y 453.511,Z 293.99,A -85,B 0,C 180,E1 -8261.944,E2 -8261.944} C_VEL
LIN {X 0,Y 453.54,Z 293.984,A -85,B 0,C 180,E1 -8264.726,E2 -8264.726} C_VEL
LIN {X 0,Y 453.559,Z 293.983,A -85,B 0,C 180,E1 -8268.379,E2 -8268.379} C_VEL
LIN {X 0,Y 453.652,Z 293.977,A -85,B 0,C 180,E1 -8271.985,E2 -8271.985} C_VEL
LIN {X 0,Y 453.666,Z 293.967,A -85,B 0,C 180,E1 -8274.667,E2 -8274.667} C_VEL
LIN {X 0,Y 453.744,Z 293.959,A -85,B 0,C 180,E1 -8277.337,E2 -8277.337} C_VEL
LIN {X 0,Y 453.822,Z 293.951,A -85,B 0,C 180,E1 -8280,E2 -8280} C_VEL
LIN {X 0,Y 453.744,Z 293.96,A -85,B 0,C 180,E1 -8282.663,E2 -8282.663} C_VEL
LIN {X 0,Y 453.668,Z 293.969,A -85,B 0,C 180,E1 -8286.225,E2 -8286.225} C_VEL
LIN {X 0,Y 453.591,Z 293.979,A -85,B 0,C 180,E1 -8288.913,E2 -8288.913} C_VEL
LIN {X 0,Y 453.564,Z 293.987,A -85,B 0,C 180,E1 -8292.529,E2 -8292.529} C_VEL
LIN {X 0,Y 453.545,Z 293.985,A -85,B 0,C 180,E1 -8296.196,E2 -8296.196} C_VEL
LIN {X 0,Y 453.52,Z 293.99,A -85,B 0,C 180,E1 -8299.04,E2 -8299.04} C_VEL
LIN {X 0,Y 453.477,Z 293.99,A -85,B 0,C 180,E1 -8301.836,E2 -8301.836} C_VEL
LIN {X 0,Y 453.507,Z 293.993,A -85,B 0,C 180,E1 -8304.735,E2 -8304.735} C_VEL
LIN {X 0,Y 453.533,Z 293.987,A -85,B 0,C 180,E1 -8307.96,E2 -8307.96} C_VEL
LIN {X 0,Y 453.465,Z 293.997,A -85,B 0,C 180,E1 -8311.525,E2 -8311.525} C_VEL
LIN {X 0,Y 453.483,Z 293.993,A -85,B 0,C 180,E1 -8314.776,E2 -8314.776} C_VEL
LIN {X 0,Y 453.464,Z 293.995,A -85,B 0,C 180,E1 -8318.312,E2 -8318.312} C_VEL
LIN {X 0,Y 453.495,Z 293.991,A -85,B 0,C 180,E1 -8320.609,E2 -8320.609} C_VEL
LIN {X 0,Y 453.456,Z 294.002,A -85,B 0,C 180,E1 -8323.244,E2 -8323.244} C_VEL
LIN {X 0,Y 453.465,Z 293.999,A -85,B 0,C 180,E1 -8325.779,E2 -8325.779} C_VEL
LIN {X 0,Y 453.481,Z 293.995,A -85,B 0,C 180,E1 -8328.209,E2 -8328.209} C_VEL
LIN {X 0,Y 453.489,Z 293.989,A -85,B 0,C 180,E1 -8330.794,E2 -8330.794} C_VEL
LIN {X 0,Y 453.456,Z 293.998,A -85,B 0,C 180,E1 -8333.917,E2 -8333.917} C_VEL
LIN {X 0,Y 453.485,Z 293.992,A -85,B 0,C 180,E1 -8337.151,E2 -8337.151} C_VEL
LIN {X 0,Y 453.477,Z 293.998,A -85,B 0,C 180,E1 -8340.268,E2 -8340.268} C_VEL
LIN {X 0,Y 453.593,Z 294.183,A -85,B 0,C 180,E1 -8343.345,E2 -8343.345} C_VEL
LIN {X 0,Y 455.884,Z 305.667,A -85,B 0,C 180,E1 -8345.637,E2 -8345.637} C_VEL
LIN {X 0,Y 456.104,Z 309.629,A -85,B 0,C 180,E1 -8346.382,E2 -8346.382} C_VEL
LIN {X 0,Y 455.163,Z 327.893,A -85,B 0,C 180,E1 -8349.67,E2 -8349.67} C_VEL
LIN {X 0,Y 454.41,Z 342.817,A -85,B 0,C 180,E1 -8352.311,E2 -8352.311} C_VEL
LIN {X 0,Y 457.787,Z 363.691,A -85,B 0,C 180,E1 -8352.8,E2 -8352.8} C_VEL
LIN {X 0,Y 457.034,Z 451.273,A -85,B 0,C 180,E1 -8354.217,E2 -8354.217} C_VEL
LIN {X 0,Y 456.626,Z 464.488,A -85,B 0,C 180,E1 -8354.603,E2 -8354.603} C_VEL
LIN {X 0,Y 456.065,Z 477.187,A -85,B 0,C 180,E1 -8355.155,E2 -8355.155} C_VEL
LIN {X 0,Y 455.527,Z 488.497,A -85,B 0,C 180,E1 -8355.822,E2 -8355.822} C_VEL
LIN {X 0,Y 454.95,Z 500.121,A -85,B 0,C 180,E1 -8356.71,E2 -8356.71} C_VEL
LIN {X 0,Y 454.388,Z 510.695,A -85,B 0,C 180,E1 -8357.721,E2 -8357.721} C_VEL
LIN {X 0,Y 453.818,Z 520.186,A -85,B 0,C 180,E1 -8358.838,E2 -8358.838} C_VEL
LIN {X 0,Y 453.296,Z 529.333,A -85,B 0,C 180,E1 -8360.18,E2 -8360.18} C_VEL
LIN {X 0,Y 452.95,Z 536.716,A -85,B 0,C 180,E1 -8361.523,E2 -8361.523} C_VEL
LIN {X 0,Y 452.716,Z 542.648,A -85,B 0,C 180,E1 -8362.865,E2 -8362.865} C_VEL
LIN {X 0,Y 452.557,Z 547.337,A -85,B 0,C 180,E1 -8364.206,E2 -8364.206} C_VEL
LIN {X 0,Y 452.487,Z 550.918,A -85,B 0,C 180,E1 -8365.545,E2 -8365.545} C_VEL
LIN {X 0,Y 452.482,Z 552.758,A -85,B 0,C 180,E1 -8366.437,E2 -8366.437} C_VEL
LIN {X 0,Y 452.508,Z 554.141,A -85,B 0,C 180,E1 -8367.329,E2 -8367.329} C_VEL
LIN {X 0,Y 452.43,Z 555.725,A -85,B 0,C 180,E1 -8369.109,E2 -8369.109} C_VEL
LIN {X 0,Y 452.465,Z 555.92,A -85,B 0,C 180,E1 -8369.999,E2 -8369.999} C_VEL
LIN {X 0,Y 452.456,Z 555.063,A -85,B 0,C 180,E1 -8371.78,E2 -8371.78} C_VEL
LIN {X 0,Y 452.507,Z 554.053,A -85,B 0,C 180,E1 -8372.67,E2 -8372.67} C_VEL
LIN {X 0,Y 452.483,Z 552.622,A -85,B 0,C 180,E1 -8373.561,E2 -8373.561} C_VEL
LIN {X 0,Y 452.545,Z 549.645,A -85,B 0,C 180,E1 -8374.899,E2 -8374.899} C_VEL
LIN {X 0,Y 452.61,Z 545.053,A -85,B 0,C 180,E1 -8376.395,E2 -8376.395} C_VEL
LIN {X 0,Y 452.84,Z 538.383,A -85,B 0,C 180,E1 -8378.028,E2 -8378.028} C_VEL
LIN {X 0,Y 453.127,Z 531.372,A -85,B 0,C 180,E1 -8379.372,E2 -8379.372} C_VEL
LIN {X 0,Y 453.55,Z 522.578,A -85,B 0,C 180,E1 -8380.716,E2 -8380.716} C_VEL
LIN {X 0,Y 454.13,Z 512.591,A -85,B 0,C 180,E1 -8381.945,E2 -8381.945} C_VEL
LIN {X 0,Y 454.635,Z 502.31,A -85,B 0,C 180,E1 -8382.962,E2 -8382.962} C_VEL
LIN {X 0,Y 455.153,Z 491.124,A -85,B 0,C 180,E1 -8383.846,E2 -8383.846} C_VEL
LIN {X 0,Y 455.675,Z 479.425,A -85,B 0,C 180,E1 -8384.571,E2 -8384.571} C_VEL
LIN {X 0,Y 456.197,Z 466.767,A -85,B 0,C 180,E1 -8385.153,E2 -8385.153} C_VEL
LIN {X 0,Y 456.59,Z 454.456,A -85,B 0,C 180,E1 -8385.54,E2 -8385.54} C_VEL
LIN {X 0,Y 456.86,Z 435.984,A -85,B 0,C 180,E1 -8385.874,E2 -8385.874} C_VEL
LIN {X 0,Y 457.322,Z 363.49,A -85,B 0,C 180,E1 -8387.021,E2 -8387.021} C_VEL
LIN {X 0,Y 454.26,Z 343.046,A -85,B 0,C 180,E1 -8387.465,E2 -8387.465} C_VEL
LIN {X 0,Y 454.978,Z 326.713,A -85,B 0,C 180,E1 -8390.337,E2 -8390.337} C_VEL
LIN {X 0,Y 455.829,Z 308.195,A -85,B 0,C 180,E1 -8393.632,E2 -8393.632} C_VEL
LIN {X 0,Y 455.456,Z 303.85,A -85,B 0,C 180,E1 -8394.438,E2 -8394.438} C_VEL
LIN {X 0,Y 453.545,Z 293.991,A -85,B 0,C 180,E1 -8396.375,E2 -8396.375} C_VEL
LIN {X 0,Y 453.509,Z 293.994,A -85,B 0,C 180,E1 -8398.711,E2 -8398.711} C_VEL
LIN {X 0,Y 453.461,Z 293.999,A -85,B 0,C 180,E1 -8401.798,E2 -8401.798} C_VEL
LIN {X 0,Y 453.478,Z 293.993,A -85,B 0,C 180,E1 -8404.988,E2 -8404.988} C_VEL
LIN {X 0,Y 453.456,Z 294.004,A -85,B 0,C 180,E1 -8408.311,E2 -8408.311} C_VEL
LIN {X 0,Y 453.489,Z 293.996,A -85,B 0,C 180,E1 -8410.608,E2 -8410.608} C_VEL
LIN {X 0,Y 453.45,Z 293.996,A -85,B 0,C 180,E1 -8413.243,E2 -8413.243} C_VEL
LIN {X 0,Y 453.467,Z 293.995,A -85,B 0,C 180,E1 -8415.779,E2 -8415.779} C_VEL
LIN {X 0,Y 453.476,Z 293.997,A -85,B 0,C 180,E1 -8418.209,E2 -8418.209} C_VEL
LIN {X 0,Y 453.509,Z 293.995,A -85,B 0,C 180,E1 -8420.789,E2 -8420.789} C_VEL
LIN {X 0,Y 453.45,Z 293.996,A -85,B 0,C 180,E1 -8423.917,E2 -8423.917} C_VEL
LIN {X 0,Y 453.476,Z 293.997,A -85,B 0,C 180,E1 -8427.151,E2 -8427.151} C_VEL
LIN {X 0,Y 453.506,Z 293.99,A -85,B 0,C 180,E1 -8430.27,E2 -8430.27} C_VEL
LIN {X 0,Y 453.506,Z 293.993,A -85,B 0,C 180,E1 -8433.294,E2 -8433.294} C_VEL
LIN {X 0,Y 453.495,Z 293.991,A -85,B 0,C 180,E1 -8436.238,E2 -8436.238} C_VEL
LIN {X 0,Y 453.474,Z 294.002,A -85,B 0,C 180,E1 -8439.117,E2 -8439.117} C_VEL
LIN {X 0,Y 453.502,Z 293.99,A -85,B 0,C 180,E1 -8441.944,E2 -8441.944} C_VEL
LIN {X 0,Y 453.532,Z 293.988,A -85,B 0,C 180,E1 -8444.726,E2 -8444.726} C_VEL
LIN {X 0,Y 453.552,Z 293.983,A -85,B 0,C 180,E1 -8448.379,E2 -8448.379} C_VEL
LIN {X 0,Y 453.642,Z 293.974,A -85,B 0,C 180,E1 -8451.985,E2 -8451.985} C_VEL
LIN {X 0,Y 453.661,Z 293.97,A -85,B 0,C 180,E1 -8454.667,E2 -8454.667} C_VEL
LIN {X 0,Y 453.755,Z 293.963,A -85,B 0,C 180,E1 -8457.337,E2 -8457.337} C_VEL
LIN {X 0,Y 453.813,Z 293.955,A -85,B 0,C 180,E1 -8460,E2 -8460} C_VEL
LIN {X 0,Y 453.756,Z 293.958,A -85,B 0,C 180,E1 -8462.663,E2 -8462.663} C_VEL
LIN {X 0,Y 453.641,Z 293.976,A -85,B 0,C 180,E1 -8466.226,E2 -8466.226} C_VEL
LIN {X 0,Y 453.582,Z 293.98,A -85,B 0,C 180,E1 -8468.914,E2 -8468.914} C_VEL
LIN {X 0,Y 453.554,Z 293.985,A -85,B 0,C 180,E1 -8472.529,E2 -8472.529} C_VEL
LIN {X 0,Y 453.547,Z 293.991,A -85,B 0,C 180,E1 -8476.196,E2 -8476.196} C_VEL
LIN {X 0,Y 453.511,Z 293.989,A -85,B 0,C 180,E1 -8479.041,E2 -8479.041} C_VEL
LIN {X 0,Y 453.467,Z 293.997,A -85,B 0,C 180,E1 -8481.837,E2 -8481.837} C_VEL
LIN {X 0,Y 453.489,Z 293.994,A -85,B 0,C 180,E1 -8484.736,E2 -8484.736} C_VEL
LIN {X 0,Y 453.52,Z 293.99,A -85,B 0,C 180,E1 -8487.959,E2 -8487.959} C_VEL
LIN {X 0,Y 453.458,Z 293.995,A -85,B 0,C 180,E1 -8491.526,E2 -8491.526} C_VEL
LIN {X 0,Y 453.48,Z 293.998,A -85,B 0,C 180,E1 -8494.778,E2 -8494.778} C_VEL
LIN {X 0,Y 453.451,Z 293.999,A -85,B 0,C 180,E1 -8498.313,E2 -8498.313} C_VEL
LIN {X 0,Y 453.464,Z 294.001,A -85,B 0,C 180,E1 -8500.612,E2 -8500.612} C_VEL
LIN {X 0,Y 453.454,Z 293.997,A -85,B 0,C 180,E1 -8504.223,E2 -8504.223} C_VEL
LIN {X 0,Y 453.432,Z 294.006,A -85,B 0,C 180,E1 -8507.003,E2 -8507.003} C_VEL
LIN {X 0,Y 453.466,Z 293.997,A -85,B 0,C 180,E1 -8509.414,E2 -8509.414} C_VEL
LIN {X 0,Y 453.445,Z 294.001,A -85,B 0,C 180,E1 -8512.811,E2 -8512.811} C_VEL
LIN {X 0,Y 453.465,Z 293.994,A -85,B 0,C 180,E1 -8516.088,E2 -8516.088} C_VEL
LIN {X 0,Y 453.462,Z 294.003,A -85,B 0,C 180,E1 -8519.241,E2 -8519.241} C_VEL
LIN {X 0,Y 453.471,Z 293.993,A -85,B 0,C 180,E1 -8522.294,E2 -8522.294} C_VEL
LIN {X 0,Y 453.466,Z 294.001,A -85,B 0,C 180,E1 -8525.264,E2 -8525.264} C_VEL
LIN {X 0,Y 453.48,Z 293.992,A -85,B 0,C 180,E1 -8528.416,E2 -8528.416} C_VEL
LIN {X 0,Y 453.523,Z 293.989,A -85,B 0,C 180,E1 -8531.01,E2 -8531.01} C_VEL
LIN {X 0,Y 453.57,Z 293.986,A -85,B 0,C 180,E1 -8533.881,E2 -8533.881} C_VEL
LIN {X 0,Y 453.565,Z 293.987,A -85,B 0,C 180,E1 -8537.472,E2 -8537.472} C_VEL
LIN {X 0,Y 453.555,Z 293.988,A -85,B 0,C 180,E1 -8541.087,E2 -8541.087} C_VEL
LIN {X 0,Y 453.555,Z 293.99,A -85,B 0,C 180,E1 -8541.727,E2 -8541.727} C_VEL
LIN {X 0,Y 453.313,Z 294.326,A -85,B 0,C 180,E1 -8542.218,E2 -8542.218} C_VEL
LIN {X 0,Y 452.229,Z 295.838,A -85,B 0,C 180,E1 -8542.927,E2 -8542.927} C_VEL
LIN {X 0,Y 450.706,Z 298.194,A -85,B 0,C 180,E1 -8543.593,E2 -8543.593} C_VEL
LIN {X 0,Y 448.654,Z 302.219,A -85,B 0,C 180,E1 -8544.461,E2 -8544.461} C_VEL
LIN {X 0,Y 447.577,Z 306.574,A -85,B 0,C 180,E1 -8545.33,E2 -8545.33} C_VEL
LIN {X 0,Y 447.46,Z 311.628,A -85,B 0,C 180,E1 -8546.371,E2 -8546.371} C_VEL
LIN {X 0,Y 450.793,Z 329.021,A -85,B 0,C 180,E1 -8546.778,E2 -8546.778} C_VEL
LIN {X 0,Y 449.894,Z 419.066,A -85,B 0,C 180,E1 -8548.238,E2 -8548.238} C_VEL
LIN {X 0,Y 449.574,Z 432.125,A -85,B 0,C 180,E1 -8548.629,E2 -8548.629} C_VEL
LIN {X 0,Y 449.187,Z 445.234,A -85,B 0,C 180,E1 -8549.216,E2 -8549.216} C_VEL
LIN {X 0,Y 448.728,Z 456.301,A -85,B 0,C 180,E1 -8549.888,E2 -8549.888} C_VEL
LIN {X 0,Y 448.16,Z 467.81,A -85,B 0,C 180,E1 -8550.787,E2 -8550.787} C_VEL
LIN {X 0,Y 447.521,Z 478.203,A -85,B 0,C 180,E1 -8551.801,E2 -8551.801} C_VEL
LIN {X 0,Y 447.01,Z 487.547,A -85,B 0,C 180,E1 -8552.93,E2 -8552.93} C_VEL
LIN {X 0,Y 446.498,Z 496.571,A -85,B 0,C 180,E1 -8554.288,E2 -8554.288} C_VEL
LIN {X 0,Y 446.088,Z 503.86,A -85,B 0,C 180,E1 -8555.651,E2 -8555.651} C_VEL
LIN {X 0,Y 445.906,Z 508.841,A -85,B 0,C 180,E1 -8556.803,E2 -8556.803} C_VEL
LIN {X 0,Y 445.696,Z 513.587,A -85,B 0,C 180,E1 -8558.159,E2 -8558.159} C_VEL
LIN {X 0,Y 445.506,Z 517.28,A -85,B 0,C 180,E1 -8559.535,E2 -8559.535} C_VEL
LIN {X 0,Y 445.424,Z 519.942,A -85,B 0,C 180,E1 -8560.915,E2 -8560.915} C_VEL
LIN {X 0,Y 445.377,Z 521.32,A -85,B 0,C 180,E1 -8561.942,E2 -8561.942} C_VEL
LIN {X 0,Y 445.282,Z 522.414,A -85,B 0,C 180,E1 -8563.695,E2 -8563.695} C_VEL
LIN {X 0,Y 445.285,Z 522.409,A -85,B 0,C 180,E1 -8564.628,E2 -8564.628} C_VEL
LIN {X 0,Y 445.324,Z 521.892,A -85,B 0,C 180,E1 -8565.7,E2 -8565.7} C_VEL
LIN {X 0,Y 445.369,Z 519.823,A -85,B 0,C 180,E1 -8567.447,E2 -8567.447} C_VEL
LIN {X 0,Y 445.564,Z 517.066,A -85,B 0,C 180,E1 -8568.844,E2 -8568.844} C_VEL
LIN {X 0,Y 445.784,Z 513.089,A -85,B 0,C 180,E1 -8570.295,E2 -8570.295} C_VEL
LIN {X 0,Y 446.09,Z 507.388,A -85,B 0,C 180,E1 -8571.863,E2 -8571.863} C_VEL
LIN {X 0,Y 446.52,Z 499.982,A -85,B 0,C 180,E1 -8573.418,E2 -8573.418} C_VEL
LIN {X 0,Y 447.063,Z 491.416,A -85,B 0,C 180,E1 -8574.843,E2 -8574.843} C_VEL
LIN {X 0,Y 447.63,Z 482.087,A -85,B 0,C 180,E1 -8576.08,E2 -8576.08} C_VEL
LIN {X 0,Y 448.267,Z 471.905,A -85,B 0,C 180,E1 -8577.17,E2 -8577.17} C_VEL
LIN {X 0,Y 448.859,Z 462.14,A -85,B 0,C 180,E1 -8578.017,E2 -8578.017} C_VEL
LIN {X 0,Y 449.449,Z 450.576,A -85,B 0,C 180,E1 -8578.819,E2 -8578.819} C_VEL
LIN {X 0,Y 449.877,Z 439.333,A -85,B 0,C 180,E1 -8579.414,E2 -8579.414} C_VEL
LIN {X 0,Y 450.228,Z 426.524,A -85,B 0,C 180,E1 -8579.904,E2 -8579.904} C_VEL
LIN {X 0,Y 450.445,Z 413.781,A -85,B 0,C 180,E1 -8580.211,E2 -8580.211} C_VEL
LIN {X 0,Y 451.402,Z 328.612,A -85,B 0,C 180,E1 -8581.586,E2 -8581.586} C_VEL
LIN {X 0,Y 447.835,Z 311.498,A -85,B 0,C 180,E1 -8582.066,E2 -8582.066} C_VEL
LIN {X 0,Y 447.88,Z 301.912,A -85,B 0,C 180,E1 -8584.019,E2 -8584.019} C_VEL
LIN {X 0,Y 446.429,Z 294.878,A -85,B 0,C 180,E1 -8585.585,E2 -8585.585} C_VEL
LIN {X 0,Y 446.44,Z 294.873,A -85,B 0,C 180,E1 -8589.028,E2 -8589.028} C_VEL
LIN {X 0,Y 446.436,Z 294.878,A -85,B 0,C 180,E1 -8592.277,E2 -8592.277} C_VEL
LIN {X 0,Y 446.453,Z 294.874,A -85,B 0,C 180,E1 -8595.104,E2 -8595.104} C_VEL
LIN {X 0,Y 446.43,Z 294.882,A -85,B 0,C 180,E1 -8598.609,E2 -8598.609} C_VEL
LIN {X 0,Y 446.461,Z 294.868,A -85,B 0,C 180,E1 -8600.974,E2 -8600.974} C_VEL
LIN {X 0,Y 446.42,Z 294.876,A -85,B 0,C 180,E1 -8604.374,E2 -8604.374} C_VEL
LIN {X 0,Y 446.423,Z 294.874,A -85,B 0,C 180,E1 -8607.638,E2 -8607.638} C_VEL
LIN {X 0,Y 446.449,Z 294.871,A -85,B 0,C 180,E1 -8610.79,E2 -8610.79} C_VEL
LIN {X 0,Y 446.479,Z 294.865,A -85,B 0,C 180,E1 -8613.848,E2 -8613.848} C_VEL
LIN {X 0,Y 446.429,Z 294.873,A -85,B 0,C 180,E1 -8616.823,E2 -8616.823} C_VEL
LIN {X 0,Y 446.444,Z 294.87,A -85,B 0,C 180,E1 -8619.737,E2 -8619.737} C_VEL
LIN {X 0,Y 446.462,Z 294.866,A -85,B 0,C 180,E1 -8622.597,E2 -8622.597} C_VEL
LIN {X 0,Y 446.47,Z 294.867,A -85,B 0,C 180,E1 -8625.412,E2 -8625.412} C_VEL
LIN {X 0,Y 446.518,Z 294.862,A -85,B 0,C 180,E1 -8628.193,E2 -8628.193} C_VEL
LIN {X 0,Y 446.6,Z 294.855,A -85,B 0,C 180,E1 -8631.858,E2 -8631.858} C_VEL
LIN {X 0,Y 446.641,Z 294.842,A -85,B 0,C 180,E1 -8634.582,E2 -8634.582} C_VEL
LIN {X 0,Y 446.663,Z 294.846,A -85,B 0,C 180,E1 -8638.197,E2 -8638.197} C_VEL
LIN {X 0,Y 446.792,Z 294.826,A -85,B 0,C 180,E1 -8640,E2 -8640} C_VEL
LIN {X 0,Y 446.691,Z 294.838,A -85,B 0,C 180,E1 -8642.705,E2 -8642.705} C_VEL
LIN {X 0,Y 446.638,Z 294.844,A -85,B 0,C 180,E1 -8646.324,E2 -8646.324} C_VEL
LIN {X 0,Y 446.536,Z 294.857,A -85,B 0,C 180,E1 -8649.055,E2 -8649.055} C_VEL
LIN {X 0,Y 446.522,Z 294.863,A -85,B 0,C 180,E1 -8652.73,E2 -8652.73} C_VEL
LIN {X 0,Y 446.496,Z 294.863,A -85,B 0,C 180,E1 -8656.228,E2 -8656.228} C_VEL
LIN {X 0,Y 446.469,Z 294.866,A -85,B 0,C 180,E1 -8659.303,E2 -8659.303} C_VEL
LIN {X 0,Y 446.418,Z 294.872,A -85,B 0,C 180,E1 -8662.2,E2 -8662.2} C_VEL
LIN {X 0,Y 446.45,Z 294.866,A -85,B 0,C 180,E1 -8665.153,E2 -8665.153} C_VEL
LIN {X 0,Y 446.485,Z 294.866,A -85,B 0,C 180,E1 -8668.179,E2 -8668.179} C_VEL
LIN {X 0,Y 446.418,Z 294.873,A -85,B 0,C 180,E1 -8671.775,E2 -8671.775} C_VEL
LIN {X 0,Y 446.423,Z 294.87,A -85,B 0,C 180,E1 -8674.524,E2 -8674.524} C_VEL
LIN {X 0,Y 446.415,Z 294.873,A -85,B 0,C 180,E1 -8678.079,E2 -8678.079} C_VEL
LIN {X 0,Y 446.428,Z 294.874,A -85,B 0,C 180,E1 -8680.918,E2 -8680.918} C_VEL
LIN {X 0,Y 446.401,Z 294.879,A -85,B 0,C 180,E1 -8683.846,E2 -8683.846} C_VEL
LIN {X 0,Y 446.399,Z 294.876,A -85,B 0,C 180,E1 -8686.404,E2 -8686.404} C_VEL
LIN {X 0,Y 446.428,Z 294.875,A -85,B 0,C 180,E1 -8689.082,E2 -8689.082} C_VEL
LIN {X 0,Y 446.41,Z 294.879,A -85,B 0,C 180,E1 -8692.121,E2 -8692.121} C_VEL
LIN {X 0,Y 446.432,Z 294.877,A -85,B 0,C 180,E1 -8695.477,E2 -8695.477} C_VEL
LIN {X 0,Y 446.418,Z 294.873,A -85,B 0,C 180,E1 -8698.7,E2 -8698.7} C_VEL
LIN {X 0,Y 446.488,Z 294.871,A -85,B 0,C 180,E1 -8701.821,E2 -8701.821} C_VEL
LIN {X 0,Y 446.545,Z 295.075,A -85,B 0,C 180,E1 -8703.071,E2 -8703.071} C_VEL
LIN {X 0,Y 449.076,Z 307.713,A -85,B 0,C 180,E1 -8705.642,E2 -8705.642} C_VEL
LIN {X 0,Y 449.1,Z 313.473,A -85,B 0,C 180,E1 -8706.725,E2 -8706.725} C_VEL
LIN {X 0,Y 448.036,Z 332.064,A -85,B 0,C 180,E1 -8710.113,E2 -8710.113} C_VEL
LIN {X 0,Y 447.481,Z 342.465,A -85,B 0,C 180,E1 -8711.985,E2 -8711.985} C_VEL
LIN {X 0,Y 451.105,Z 365.037,A -85,B 0,C 180,E1 -8712.534,E2 -8712.534} C_VEL
LIN {X 0,Y 450.275,Z 451.034,A -85,B 0,C 180,E1 -8713.945,E2 -8713.945} C_VEL
LIN {X 0,Y 449.844,Z 464.238,A -85,B 0,C 180,E1 -8714.336,E2 -8714.336} C_VEL
LIN {X 0,Y 449.227,Z 477.49,A -85,B 0,C 180,E1 -8714.924,E2 -8714.924} C_VEL
LIN {X 0,Y 448.665,Z 488.634,A -85,B 0,C 180,E1 -8715.601,E2 -8715.601} C_VEL
LIN {X 0,Y 448.02,Z 500.148,A -85,B 0,C 180,E1 -8716.499,E2 -8716.499} C_VEL
LIN {X 0,Y 447.437,Z 510.668,A -85,B 0,C 180,E1 -8717.527,E2 -8717.527} C_VEL
LIN {X 0,Y 446.846,Z 520.097,A -85,B 0,C 180,E1 -8718.661,E2 -8718.661} C_VEL
LIN {X 0,Y 446.277,Z 529.198,A -85,B 0,C 180,E1 -8720.024,E2 -8720.024} C_VEL
LIN {X 0,Y 445.884,Z 536.553,A -85,B 0,C 180,E1 -8721.388,E2 -8721.388} C_VEL
LIN {X 0,Y 445.633,Z 542.467,A -85,B 0,C 180,E1 -8722.751,E2 -8722.751} C_VEL
LIN {X 0,Y 445.47,Z 546.636,A -85,B 0,C 180,E1 -8723.955,E2 -8723.955} C_VEL
LIN {X 0,Y 445.412,Z 550.703,A -85,B 0,C 180,E1 -8725.474,E2 -8725.474} C_VEL
LIN {X 0,Y 445.38,Z 552.526,A -85,B 0,C 180,E1 -8726.381,E2 -8726.381} C_VEL
LIN {X 0,Y 445.433,Z 553.903,A -85,B 0,C 180,E1 -8727.286,E2 -8727.286} C_VEL
LIN {X 0,Y 445.34,Z 555.472,A -85,B 0,C 180,E1 -8729.095,E2 -8729.095} C_VEL
LIN {X 0,Y 445.371,Z 555.652,A -85,B 0,C 180,E1 -8729.999,E2 -8729.999} C_VEL
LIN {X 0,Y 445.374,Z 554.78,A -85,B 0,C 180,E1 -8731.808,E2 -8731.808} C_VEL
LIN {X 0,Y 445.432,Z 553.761,A -85,B 0,C 180,E1 -8732.712,E2 -8732.712} C_VEL
LIN {X 0,Y 445.383,Z 552.313,A -85,B 0,C 180,E1 -8733.618,E2 -8733.618} C_VEL
LIN {X 0,Y 445.473,Z 549.323,A -85,B 0,C 180,E1 -8734.977,E2 -8734.977} C_VEL
LIN {X 0,Y 445.556,Z 543.809,A -85,B 0,C 180,E1 -8736.748,E2 -8736.748} C_VEL
LIN {X 0,Y 445.768,Z 538.016,A -85,B 0,C 180,E1 -8738.157,E2 -8738.157} C_VEL
LIN {X 0,Y 446.07,Z 530.974,A -85,B 0,C 180,E1 -8739.521,E2 -8739.521} C_VEL
LIN {X 0,Y 446.544,Z 522.148,A -85,B 0,C 180,E1 -8740.886,E2 -8740.886} C_VEL
LIN {X 0,Y 447.151,Z 512.126,A -85,B 0,C 180,E1 -8742.134,E2 -8742.134} C_VEL
LIN {X 0,Y 447.65,Z 501.775,A -85,B 0,C 180,E1 -8743.168,E2 -8743.168} C_VEL
LIN {X 0,Y 448.199,Z 490.513,A -85,B 0,C 180,E1 -8744.066,E2 -8744.066} C_VEL
LIN {X 0,Y 448.787,Z 478.715,A -85,B 0,C 180,E1 -8744.8,E2 -8744.8} C_VEL
LIN {X 0,Y 449.313,Z 465.797,A -85,B 0,C 180,E1 -8745.391,E2 -8745.391} C_VEL
LIN {X 0,Y 449.753,Z 453.128,A -85,B 0,C 180,E1 -8745.782,E2 -8745.782} C_VEL
LIN {X 0,Y 450.081,Z 426.871,A -85,B 0,C 180,E1 -8746.236,E2 -8746.236} C_VEL
LIN {X 0,Y 450.489,Z 364.205,A -85,B 0,C 180,E1 -8747.242,E2 -8747.242} C_VEL
LIN {X 0,Y 447.269,Z 342.842,A -85,B 0,C 180,E1 -8747.707,E2 -8747.707} C_VEL
LIN {X 0,Y 448.134,Z 324.955,A -85,B 0,C 180,E1 -8750.902,E2 -8750.902} C_VEL
LIN {X 0,Y 448.872,Z 309.051,A -85,B 0,C 180,E1 -8753.775,E2 -8753.775} C_VEL
LIN {X 0,Y 448.266,Z 303.812,A -85,B 0,C 180,E1 -8754.77,E2 -8754.77} C_VEL
LIN {X 0,Y 446.499,Z 294.868,A -85,B 0,C 180,E1 -8756.528,E2 -8756.528} C_VEL
LIN {X 0,Y 446.447,Z 294.873,A -85,B 0,C 180,E1 -8759.208,E2 -8759.208} C_VEL
LIN {X 0,Y 446.419,Z 294.877,A -85,B 0,C 180,E1 -8762.361,E2 -8762.361} C_VEL
LIN {X 0,Y 446.417,Z 294.873,A -85,B 0,C 180,E1 -8765.625,E2 -8765.625} C_VEL
LIN {X 0,Y 446.434,Z 294.871,A -85,B 0,C 180,E1 -8769.027,E2 -8769.027} C_VEL
LIN {X 0,Y 446.429,Z 294.877,A -85,B 0,C 180,E1 -8772.276,E2 -8772.276} C_VEL
LIN {X 0,Y 446.45,Z 294.869,A -85,B 0,C 180,E1 -8775.102,E2 -8775.102} C_VEL
LIN {X 0,Y 446.423,Z 294.88,A -85,B 0,C 180,E1 -8778.608,E2 -8778.608} C_VEL
LIN {X 0,Y 446.455,Z 294.871,A -85,B 0,C 180,E1 -8780.974,E2 -8780.974} C_VEL
LIN {X 0,Y 446.414,Z 294.876,A -85,B 0,C 180,E1 -8784.373,E2 -8784.373} C_VEL
LIN {X 0,Y 446.422,Z 294.872,A -85,B 0,C 180,E1 -8787.638,E2 -8787.638} C_VEL
LIN {X 0,Y 446.462,Z 294.874,A -85,B 0,C 180,E1 -8790.791,E2 -8790.791} C_VEL
LIN {X 0,Y 446.469,Z 294.866,A -85,B 0,C 180,E1 -8793.848,E2 -8793.848} C_VEL
LIN {X 0,Y 446.42,Z 294.877,A -85,B 0,C 180,E1 -8796.823,E2 -8796.823} C_VEL
LIN {X 0,Y 446.435,Z 294.871,A -85,B 0,C 180,E1 -8799.737,E2 -8799.737} C_VEL
LIN {X 0,Y 446.454,Z 294.869,A -85,B 0,C 180,E1 -8802.597,E2 -8802.597} C_VEL
LIN {X 0,Y 446.463,Z 294.873,A -85,B 0,C 180,E1 -8805.412,E2 -8805.412} C_VEL
LIN {X 0,Y 446.509,Z 294.861,A -85,B 0,C 180,E1 -8808.193,E2 -8808.193} C_VEL
LIN {X 0,Y 446.591,Z 294.854,A -85,B 0,C 180,E1 -8811.858,E2 -8811.858} C_VEL
LIN {X 0,Y 446.635,Z 294.845,A -85,B 0,C 180,E1 -8814.583,E2 -8814.583} C_VEL
LIN {X 0,Y 446.699,Z 294.841,A -85,B 0,C 180,E1 -8817.295,E2 -8817.295} C_VEL
LIN {X 0,Y 446.783,Z 294.831,A -85,B 0,C 180,E1 -8820,E2 -8820} C_VEL
LIN {X 0,Y 446.7,Z 294.837,A -85,B 0,C 180,E1 -8822.705,E2 -8822.705} C_VEL
LIN {X 0,Y 446.609,Z 294.851,A -85,B 0,C 180,E1 -8826.324,E2 -8826.324} C_VEL
LIN {X 0,Y 446.528,Z 294.858,A -85,B 0,C 180,E1 -8829.056,E2 -8829.056} C_VEL
LIN {X 0,Y 446.512,Z 294.861,A -85,B 0,C 180,E1 -8832.73,E2 -8832.73} C_VEL
LIN {X 0,Y 446.51,Z 294.867,A -85,B 0,C 180,E1 -8836.238,E2 -8836.238} C_VEL
LIN {X 0,Y 446.46,Z 294.867,A -85,B 0,C 180,E1 -8839.304,E2 -8839.304} C_VEL
LIN {X 0,Y 446.409,Z 294.881,A -85,B 0,C 180,E1 -8842.2,E2 -8842.2} C_VEL
LIN {X 0,Y 446.432,Z 294.871,A -85,B 0,C 180,E1 -8845.154,E2 -8845.154} C_VEL
LIN {X 0,Y 446.477,Z 294.87,A -85,B 0,C 180,E1 -8848.179,E2 -8848.179} C_VEL
LIN {X 0,Y 446.411,Z 294.873,A -85,B 0,C 180,E1 -8851.776,E2 -8851.776} C_VEL
LIN {X 0,Y 446.422,Z 294.879,A -85,B 0,C 180,E1 -8854.524,E2 -8854.524} C_VEL
LIN {X 0,Y 446.405,Z 294.875,A -85,B 0,C 180,E1 -8858.079,E2 -8858.079} C_VEL
LIN {X 0,Y 446.404,Z 294.875,A -85,B 0,C 180,E1 -8861.394,E2 -8861.394} C_VEL
LIN {X 0,Y 446.444,Z 294.874,A -85,B 0,C 180,E1 -8865.105,E2 -8865.105} C_VEL
LIN {X 0,Y 446.401,Z 294.878,A -85,B 0,C 180,E1 -8868.607,E2 -8868.607} C_VEL
LIN {X 0,Y 446.406,Z 294.874,A -85,B 0,C 180,E1 -8871.923,E2 -8871.923} C_VEL
LIN {X 0,Y 446.419,Z 294.876,A -85,B 0,C 180,E1 -8875.477,E2 -8875.477} C_VEL
LIN {X 0,Y 446.409,Z 294.875,A -85,B 0,C 180,E1 -8878.7,E2 -8878.7} C_VEL
LIN {X 0,Y 446.421,Z 294.874,A -85,B 0,C 180,E1 -8881.837,E2 -8881.837} C_VEL
LIN {X 0,Y 446.418,Z 294.874,A -85,B 0,C 180,E1 -8884.846,E2 -8884.846} C_VEL
LIN {X 0,Y 446.448,Z 294.869,A -85,B 0,C 180,E1 -8888.246,E2 -8888.246} C_VEL
LIN {X 0,Y 446.449,Z 294.876,A -85,B 0,C 180,E1 -8891.65,E2 -8891.65} C_VEL
LIN {X 0,Y 446.505,Z 294.861,A -85,B 0,C 180,E1 -8894.481,E2 -8894.481} C_VEL
LIN {X 0,Y 446.5,Z 294.865,A -85,B 0,C 180,E1 -8898.193,E2 -8898.193} C_VEL
LIN {X 0,Y 446.512,Z 294.869,A -85,B 0,C 180,E1 -8901.734,E2 -8901.734} C_VEL
LIN {X 0,Y 446.579,Z 295.036,A -85,B 0,C 180,E1 -8902.868,E2 -8902.868} C_VEL
LIN {X 0,Y 447.663,Z 301.932,A -85,B 0,C 180,E1 -8904.37,E2 -8904.37} C_VEL
LIN {X 0,Y 447.577,Z 306.574,A -85,B 0,C 180,E1 -8905.33,E2 -8905.33} C_VEL
LIN {X 0,Y 447.33,Z 309.068,A -85,B 0,C 180,E1 -8905.704,E2 -8905.704} C_VEL
LIN {X 0,Y 446.599,Z 313.931,A -85,B 0,C 180,E1 -8906.105,E2 -8906.105} C_VEL
LIN {X 0,Y 445.683,Z 319.461,A -85,B 0,C 180,E1 -8906.349,E2 -8906.349} C_VEL
LIN {X 0,Y 444.482,Z 327.65,A -85,B 0,C 180,E1 -8906.525,E2 -8906.525} C_VEL
LIN {X 0,Y 443.905,Z 335.973,A -85,B 0,C 180,E1 -8906.645,E2 -8906.645} C_VEL
LIN {X 0,Y 443.03,Z 419.515,A -85,B 0,C 180,E1 -8908.023,E2 -8908.023} C_VEL
LIN {X 0,Y 442.694,Z 432.223,A -85,B 0,C 180,E1 -8908.409,E2 -8908.409} C_VEL
LIN {X 0,Y 442.304,Z 444.824,A -85,B 0,C 180,E1 -8908.976,E2 -8908.976} C_VEL
LIN {X 0,Y 441.822,Z 456.08,A -85,B 0,C 180,E1 -8909.659,E2 -8909.659} C_VEL
LIN {X 0,Y 441.225,Z 467.685,A -85,B 0,C 180,E1 -8910.571,E2 -8910.571} C_VEL
LIN {X 0,Y 440.571,Z 478.14,A -85,B 0,C 180,E1 -8911.6,E2 -8911.6} C_VEL
LIN {X 0,Y 440.038,Z 487.553,A -85,B 0,C 180,E1 -8912.747,E2 -8912.747} C_VEL
LIN {X 0,Y 439.469,Z 496.632,A -85,B 0,C 180,E1 -8914.127,E2 -8914.127} C_VEL
LIN {X 0,Y 439.038,Z 503.957,A -85,B 0,C 180,E1 -8915.512,E2 -8915.512} C_VEL
LIN {X 0,Y 438.79,Z 510.495,A -85,B 0,C 180,E1 -8917.082,E2 -8917.082} C_VEL
LIN {X 0,Y 438.506,Z 515.742,A -85,B 0,C 180,E1 -8918.758,E2 -8918.758} C_VEL
LIN {X 0,Y 438.366,Z 518.936,A -85,B 0,C 180,E1 -8920.158,E2 -8920.158} C_VEL
LIN {X 0,Y 438.316,Z 520.525,A -85,B 0,C 180,E1 -8921.094,E2 -8921.094} C_VEL
LIN {X 0,Y 438.297,Z 521.674,A -85,B 0,C 180,E1 -8922.032,E2 -8922.032} C_VEL
LIN {X 0,Y 438.214,Z 522.394,A -85,B 0,C 180,E1 -8922.976,E2 -8922.976} C_VEL
LIN {X 0,Y 438.179,Z 522.716,A -85,B 0,C 180,E1 -8923.922,E2 -8923.922} C_VEL
LIN {X 0,Y 438.22,Z 522.637,A -85,B 0,C 180,E1 -8924.869,E2 -8924.869} C_VEL
LIN {X 0,Y 438.242,Z 522.1,A -85,B 0,C 180,E1 -8925.821,E2 -8925.821} C_VEL
LIN {X 0,Y 438.232,Z 521.143,A -85,B 0,C 180,E1 -8926.779,E2 -8926.779} C_VEL
LIN {X 0,Y 438.31,Z 519.769,A -85,B 0,C 180,E1 -8927.738,E2 -8927.738} C_VEL
LIN {X 0,Y 438.5,Z 517.264,A -85,B 0,C 180,E1 -8928.982,E2 -8928.982} C_VEL
LIN {X 0,Y 438.778,Z 512.721,A -85,B 0,C 180,E1 -8930.633,E2 -8930.633} C_VEL
LIN {X 0,Y 439.138,Z 506.285,A -85,B 0,C 180,E1 -8932.338,E2 -8932.338} C_VEL
LIN {X 0,Y 439.633,Z 499.249,A -85,B 0,C 180,E1 -8933.786,E2 -8933.786} C_VEL
LIN {X 0,Y 440.107,Z 491.751,A -85,B 0,C 180,E1 -8935.035,E2 -8935.035} C_VEL
LIN {X 0,Y 440.722,Z 482.653,A -85,B 0,C 180,E1 -8936.265,E2 -8936.265} C_VEL
LIN {X 0,Y 441.404,Z 472.292,A -85,B 0,C 180,E1 -8937.396,E2 -8937.396} C_VEL
LIN {X 0,Y 442.002,Z 462.847,A -85,B 0,C 180,E1 -8938.232,E2 -8938.232} C_VEL
LIN {X 0,Y 442.622,Z 451.574,A -85,B 0,C 180,E1 -8939.036,E2 -8939.036} C_VEL
LIN {X 0,Y 443.095,Z 440.455,A -85,B 0,C 180,E1 -8939.648,E2 -8939.648} C_VEL
LIN {X 0,Y 443.457,Z 428.021,A -85,B 0,C 180,E1 -8940.145,E2 -8940.145} C_VEL
LIN {X 0,Y 443.718,Z 414.619,A -85,B 0,C 180,E1 -8940.485,E2 -8940.485} C_VEL
LIN {X 0,Y 444.716,Z 329.474,A -85,B 0,C 180,E1 -8941.885,E2 -8941.885} C_VEL
LIN {X 0,Y 440.945,Z 311.764,A -85,B 0,C 180,E1 -8942.395,E2 -8942.395} C_VEL
LIN {X 0,Y 441.029,Z 303.776,A -85,B 0,C 180,E1 -8944.04,E2 -8944.04} C_VEL
LIN {X 0,Y 439.383,Z 295.757,A -85,B 0,C 180,E1 -8945.858,E2 -8945.858} C_VEL
LIN {X 0,Y 439.378,Z 295.753,A -85,B 0,C 180,E1 -8948.596,E2 -8948.596} C_VEL
LIN {X 0,Y 439.391,Z 295.751,A -85,B 0,C 180,E1 -8951.257,E2 -8951.257} C_VEL
LIN {X 0,Y 439.402,Z 295.756,A -85,B 0,C 180,E1 -8954.729,E2 -8954.729} C_VEL
LIN {X 0,Y 439.398,Z 295.751,A -85,B 0,C 180,E1 -8957.796,E2 -8957.796} C_VEL
LIN {X 0,Y 439.438,Z 295.744,A -85,B 0,C 180,E1 -8960.228,E2 -8960.228} C_VEL
LIN {X 0,Y 439.375,Z 295.752,A -85,B 0,C 180,E1 -8963.713,E2 -8963.713} C_VEL
LIN {X 0,Y 439.374,Z 295.755,A -85,B 0,C 180,E1 -8967.054,E2 -8967.054} C_VEL
LIN {X 0,Y 439.383,Z 295.747,A -85,B 0,C 180,E1 -8970.274,E2 -8970.274} C_VEL
LIN {X 0,Y 439.429,Z 295.746,A -85,B 0,C 180,E1 -8973.396,E2 -8973.396} C_VEL
LIN {X 0,Y 439.387,Z 295.748,A -85,B 0,C 180,E1 -8976.429,E2 -8976.429} C_VEL
LIN {X 0,Y 439.389,Z 295.754,A -85,B 0,C 180,E1 -8979.397,E2 -8979.397} C_VEL
LIN {X 0,Y 439.431,Z 295.742,A -85,B 0,C 180,E1 -8982.309,E2 -8982.309} C_VEL
LIN {X 0,Y 439.448,Z 295.743,A -85,B 0,C 180,E1 -8985.174,E2 -8985.174} C_VEL
LIN {X 0,Y 439.484,Z 295.74,A -85,B 0,C 180,E1 -8988.001,E2 -8988.001} C_VEL
LIN {X 0,Y 439.548,Z 295.731,A -85,B 0,C 180,E1 -8991.726,E2 -8991.726} C_VEL
LIN {X 0,Y 439.616,Z 295.718,A -85,B 0,C 180,E1 -8994.496,E2 -8994.496} C_VEL
LIN {X 0,Y 439.634,Z 295.722,A -85,B 0,C 180,E1 -8998.168,E2 -8998.168} C_VEL
LIN {X 0,Y 439.762,Z 295.701,A -85,B 0,C 180,E1 -9000,E2 -9000} C_VEL
LIN {X 0,Y 439.641,Z 295.717,A -85,B 0,C 180,E1 -9002.749,E2 -9002.749} C_VEL
LIN {X 0,Y 439.613,Z 295.719,A -85,B 0,C 180,E1 -9006.425,E2 -9006.425} C_VEL
LIN {X 0,Y 439.498,Z 295.733,A -85,B 0,C 180,E1 -9009.202,E2 -9009.202} C_VEL
LIN {X 0,Y 439.466,Z 295.74,A -85,B 0,C 180,E1 -9012.938,E2 -9012.938} C_VEL
LIN {X 0,Y 439.447,Z 295.74,A -85,B 0,C 180,E1 -9016.349,E2 -9016.349} C_VEL
LIN {X 0,Y 439.403,Z 295.746,A -85,B 0,C 180,E1 -9019.626,E2 -9019.626} C_VEL
LIN {X 0,Y 439.365,Z 295.755,A -85,B 0,C 180,E1 -9022.575,E2 -9022.575} C_VEL
LIN {X 0,Y 439.401,Z 295.741,A -85,B 0,C 180,E1 -9025.585,E2 -9025.585} C_VEL
LIN {X 0,Y 439.418,Z 295.751,A -85,B 0,C 180,E1 -9028.673,E2 -9028.673} C_VEL
LIN {X 0,Y 439.369,Z 295.751,A -85,B 0,C 180,E1 -9032.03,E2 -9032.03} C_VEL
LIN {X 0,Y 439.393,Z 295.753,A -85,B 0,C 180,E1 -9035.34,E2 -9035.34} C_VEL
LIN {X 0,Y 439.378,Z 295.751,A -85,B 0,C 180,E1 -9038.596,E2 -9038.596} C_VEL
LIN {X 0,Y 439.39,Z 295.753,A -85,B 0,C 180,E1 -9041.257,E2 -9041.257} C_VEL
LIN {X 0,Y 439.401,Z 295.749,A -85,B 0,C 180,E1 -9044.729,E2 -9044.729} C_VEL
LIN {X 0,Y 439.397,Z 295.752,A -85,B 0,C 180,E1 -9047.796,E2 -9047.796} C_VEL
LIN {X 0,Y 439.396,Z 295.745,A -85,B 0,C 180,E1 -9050.224,E2 -9050.224} C_VEL
LIN {X 0,Y 439.376,Z 295.753,A -85,B 0,C 180,E1 -9053.713,E2 -9053.713} C_VEL
LIN {X 0,Y 439.375,Z 295.75,A -85,B 0,C 180,E1 -9057.054,E2 -9057.054} C_VEL
LIN {X 0,Y 439.385,Z 295.753,A -85,B 0,C 180,E1 -9060.274,E2 -9060.274} C_VEL
LIN {X 0,Y 439.489,Z 295.855,A -85,B 0,C 180,E1 -9062.758,E2 -9062.758} C_VEL
LIN {X 0,Y 441.919,Z 307.733,A -85,B 0,C 180,E1 -9065.232,E2 -9065.232} C_VEL
LIN {X 0,Y 442.332,Z 312.123,A -85,B 0,C 180,E1 -9066.099,E2 -9066.099} C_VEL
LIN {X 0,Y 441.35,Z 327.752,A -85,B 0,C 180,E1 -9069.005,E2 -9069.005} C_VEL
LIN {X 0,Y 440.578,Z 342.243,A -85,B 0,C 180,E1 -9071.663,E2 -9071.663} C_VEL
LIN {X 0,Y 444.345,Z 365.259,A -85,B 0,C 180,E1 -9072.233,E2 -9072.233} C_VEL
LIN {X 0,Y 443.534,Z 450.8,A -85,B 0,C 180,E1 -9073.664,E2 -9073.664} C_VEL
LIN {X 0,Y 443.08,Z 463.987,A -85,B 0,C 180,E1 -9074.061,E2 -9074.061} C_VEL
LIN {X 0,Y 442.46,Z 476.675,A -85,B 0,C 180,E1 -9074.629,E2 -9074.629} C_VEL
LIN {X 0,Y 441.806,Z 488.768,A -85,B 0,C 180,E1 -9075.372,E2 -9075.372} C_VEL
LIN {X 0,Y 441.186,Z 498.993,A -85,B 0,C 180,E1 -9076.175,E2 -9076.175} C_VEL
LIN {X 0,Y 440.545,Z 509.603,A -85,B 0,C 180,E1 -9077.211,E2 -9077.211} C_VEL
LIN {X 0,Y 439.88,Z 520.039,A -85,B 0,C 180,E1 -9078.479,E2 -9078.479} C_VEL
LIN {X 0,Y 439.254,Z 529.103,A -85,B 0,C 180,E1 -9079.863,E2 -9079.863} C_VEL
LIN {X 0,Y 438.846,Z 536.424,A -85,B 0,C 180,E1 -9081.248,E2 -9081.248} C_VEL
LIN {X 0,Y 438.581,Z 542.306,A -85,B 0,C 180,E1 -9082.634,E2 -9082.634} C_VEL
LIN {X 0,Y 438.371,Z 546.88,A -85,B 0,C 180,E1 -9083.995,E2 -9083.995} C_VEL
LIN {X 0,Y 438.341,Z 550.494,A -85,B 0,C 180,E1 -9085.401,E2 -9085.401} C_VEL
LIN {X 0,Y 438.282,Z 552.297,A -85,B 0,C 180,E1 -9086.322,E2 -9086.322} C_VEL
LIN {X 0,Y 438.341,Z 553.666,A -85,B 0,C 180,E1 -9087.242,E2 -9087.242} C_VEL
LIN {X 0,Y 438.295,Z 554.636,A -85,B 0,C 180,E1 -9088.162,E2 -9088.162} C_VEL
LIN {X 0,Y 438.254,Z 555.219,A -85,B 0,C 180,E1 -9089.08,E2 -9089.08} C_VEL
LIN {X 0,Y 438.28,Z 555.384,A -85,B 0,C 180,E1 -9089.999,E2 -9089.999} C_VEL
LIN {X 0,Y 438.295,Z 554.496,A -85,B 0,C 180,E1 -9091.837,E2 -9091.837} C_VEL
LIN {X 0,Y 438.359,Z 553.47,A -85,B 0,C 180,E1 -9092.756,E2 -9092.756} C_VEL
LIN {X 0,Y 438.285,Z 552.004,A -85,B 0,C 180,E1 -9093.677,E2 -9093.677} C_VEL
LIN {X 0,Y 438.382,Z 548.997,A -85,B 0,C 180,E1 -9095.058,E2 -9095.058} C_VEL
LIN {X 0,Y 438.447,Z 544.923,A -85,B 0,C 180,E1 -9096.442,E2 -9096.442} C_VEL
LIN {X 0,Y 438.668,Z 538.655,A -85,B 0,C 180,E1 -9098.058,E2 -9098.058} C_VEL
LIN {X 0,Y 438.973,Z 531.824,A -85,B 0,C 180,E1 -9099.444,E2 -9099.444} C_VEL
LIN {X 0,Y 439.413,Z 523.32,A -85,B 0,C 180,E1 -9100.831,E2 -9100.831} C_VEL
LIN {X 0,Y 439.958,Z 514.557,A -85,B 0,C 180,E1 -9101.985,E2 -9101.985} C_VEL
LIN {X 0,Y 440.542,Z 504.721,A -85,B 0,C 180,E1 -9103.044,E2 -9103.044} C_VEL
LIN {X 0,Y 441.079,Z 494.448,A -85,B 0,C 180,E1 -9103.944,E2 -9103.944} C_VEL
LIN {X 0,Y 441.657,Z 482.901,A -85,B 0,C 180,E1 -9104.749,E2 -9104.749} C_VEL
LIN {X 0,Y 442.245,Z 470.934,A -85,B 0,C 180,E1 -9105.377,E2 -9105.377} C_VEL
LIN {X 0,Y 442.665,Z 457.995,A -85,B 0,C 180,E1 -9105.864,E2 -9105.864} C_VEL
LIN {X 0,Y 443.034,Z 445.994,A -85,B 0,C 180,E1 -9106.146,E2 -9106.146} C_VEL
LIN {X 0,Y 443.587,Z 364.587,A -85,B 0,C 180,E1 -9107.476,E2 -9107.476} C_VEL
LIN {X 0,Y 440.281,Z 342.492,A -85,B 0,C 180,E1 -9107.979,E2 -9107.979} C_VEL
LIN {X 0,Y 441.155,Z 325.81,A -85,B 0,C 180,E1 -9111.004,E2 -9111.004} C_VEL
LIN {X 0,Y 441.909,Z 309.9,A -85,B 0,C 180,E1 -9113.924,E2 -9113.924} C_VEL
LIN {X 0,Y 440.888,Z 302.847,A -85,B 0,C 180,E1 -9115.295,E2 -9115.295} C_VEL
LIN {X 0,Y 439.464,Z 295.745,A -85,B 0,C 180,E1 -9116.728,E2 -9116.728} C_VEL
LIN {X 0,Y 439.38,Z 295.757,A -85,B 0,C 180,E1 -9119.725,E2 -9119.725} C_VEL
LIN {X 0,Y 439.369,Z 295.751,A -85,B 0,C 180,E1 -9122.945,E2 -9122.945} C_VEL
LIN {X 0,Y 439.371,Z 295.758,A -85,B 0,C 180,E1 -9126.286,E2 -9126.286} C_VEL
LIN {X 0,Y 439.397,Z 295.749,A -85,B 0,C 180,E1 -9129.848,E2 -9129.848} C_VEL
LIN {X 0,Y 439.377,Z 295.755,A -85,B 0,C 180,E1 -9132.626,E2 -9132.626} C_VEL
LIN {X 0,Y 439.4,Z 295.747,A -85,B 0,C 180,E1 -9135.27,E2 -9135.27} C_VEL
LIN {X 0,Y 439.383,Z 295.755,A -85,B 0,C 180,E1 -9138.742,E2 -9138.742} C_VEL
LIN {X 0,Y 439.379,Z 295.749,A -85,B 0,C 180,E1 -9141.605,E2 -9141.605} C_VEL
LIN {X 0,Y 439.393,Z 295.754,A -85,B 0,C 180,E1 -9144.843,E2 -9144.843} C_VEL
LIN {X 0,Y 439.383,Z 295.749,A -85,B 0,C 180,E1 -9148.14,E2 -9148.14} C_VEL
LIN {X 0,Y 439.417,Z 295.747,A -85,B 0,C 180,E1 -9151.326,E2 -9151.326} C_VEL
LIN {X 0,Y 439.397,Z 295.748,A -85,B 0,C 180,E1 -9154.415,E2 -9154.415} C_VEL
LIN {X 0,Y 439.356,Z 295.756,A -85,B 0,C 180,E1 -9157.424,E2 -9157.424} C_VEL
LIN {X 0,Y 439.432,Z 295.744,A -85,B 0,C 180,E1 -9160.662,E2 -9160.662} C_VEL
LIN {X 0,Y 439.454,Z 295.74,A -85,B 0,C 180,E1 -9164.224,E2 -9164.224} C_VEL
LIN {X 0,Y 439.475,Z 295.738,A -85,B 0,C 180,E1 -9168.001,E2 -9168.001} C_VEL
LIN {X 0,Y 439.539,Z 295.734,A -85,B 0,C 180,E1 -9171.726,E2 -9171.726} C_VEL
LIN {X 0,Y 439.611,Z 295.72,A -85,B 0,C 180,E1 -9174.496,E2 -9174.496} C_VEL
LIN {X 0,Y 439.625,Z 295.72,A -85,B 0,C 180,E1 -9178.168,E2 -9178.168} C_VEL
LIN {X 0,Y 439.753,Z 295.706,A -85,B 0,C 180,E1 -9180,E2 -9180} C_VEL
LIN {X 0,Y 439.646,Z 295.716,A -85,B 0,C 180,E1 -9182.749,E2 -9182.749} C_VEL
LIN {X 0,Y 439.57,Z 295.726,A -85,B 0,C 180,E1 -9186.522,E2 -9186.522} C_VEL
LIN {X 0,Y 439.49,Z 295.736,A -85,B 0,C 180,E1 -9189.202,E2 -9189.202} C_VEL
LIN {X 0,Y 439.456,Z 295.739,A -85,B 0,C 180,E1 -9192.938,E2 -9192.938} C_VEL
LIN {X 0,Y 439.451,Z 295.745,A -85,B 0,C 180,E1 -9196.355,E2 -9196.355} C_VEL
LIN {X 0,Y 439.393,Z 295.749,A -85,B 0,C 180,E1 -9199.627,E2 -9199.627} C_VEL
LIN {X 0,Y 439.355,Z 295.756,A -85,B 0,C 180,E1 -9202.576,E2 -9202.576} C_VEL
LIN {X 0,Y 439.379,Z 295.749,A -85,B 0,C 180,E1 -9205.587,E2 -9205.587} C_VEL
LIN {X 0,Y 439.409,Z 295.75,A -85,B 0,C 180,E1 -9208.674,E2 -9208.674} C_VEL
LIN {X 0,Y 439.362,Z 295.753,A -85,B 0,C 180,E1 -9212.031,E2 -9212.031} C_VEL
LIN {X 0,Y 439.387,Z 295.749,A -85,B 0,C 180,E1 -9215.341,E2 -9215.341} C_VEL
LIN {X 0,Y 439.355,Z 295.759,A -85,B 0,C 180,E1 -9218.598,E2 -9218.598} C_VEL
LIN {X 0,Y 439.376,Z 295.751,A -85,B 0,C 180,E1 -9222.207,E2 -9222.207} C_VEL
LIN {X 0,Y 439.392,Z 295.751,A -85,B 0,C 180,E1 -9225.271,E2 -9225.271} C_VEL
LIN {X 0,Y 439.353,Z 295.76,A -85,B 0,C 180,E1 -9229.018,E2 -9229.018} C_VEL
LIN {X 0,Y 439.362,Z 295.753,A -85,B 0,C 180,E1 -9231.61,E2 -9231.61} C_VEL
LIN {X 0,Y 439.392,Z 295.752,A -85,B 0,C 180,E1 -9234.845,E2 -9234.845} C_VEL
LIN {X 0,Y 439.368,Z 295.75,A -85,B 0,C 180,E1 -9238.14,E2 -9238.14} C_VEL
LIN {X 0,Y 439.385,Z 295.753,A -85,B 0,C 180,E1 -9241.61,E2 -9241.61} C_VEL
LIN {X 0,Y 439.363,Z 295.751,A -85,B 0,C 180,E1 -9244.414,E2 -9244.414} C_VEL
LIN {X 0,Y 439.361,Z 295.759,A -85,B 0,C 180,E1 -9247.425,E2 -9247.425} C_VEL
LIN {X 0,Y 439.441,Z 295.741,A -85,B 0,C 180,E1 -9250.664,E2 -9250.664} C_VEL
LIN {X 0,Y 439.461,Z 295.74,A -85,B 0,C 180,E1 -9254.225,E2 -9254.225} C_VEL
LIN {X 0,Y 439.471,Z 295.742,A -85,B 0,C 180,E1 -9258.002,E2 -9258.002} C_VEL
LIN {X 0,Y 439.48,Z 295.746,A -85,B 0,C 180,E1 -9261.726,E2 -9261.726} C_VEL
LIN {X 0,Y 439.561,Z 295.936,A -85,B 0,C 180,E1 -9262.709,E2 -9262.709} C_VEL
LIN {X 0,Y 440.714,Z 303.077,A -85,B 0,C 180,E1 -9264.281,E2 -9264.281} C_VEL
LIN {X 0,Y 440.513,Z 311.836,A -85,B 0,C 180,E1 -9266.113,E2 -9266.113} C_VEL
LIN {X 0,Y 443.928,Z 329.305,A -85,B 0,C 180,E1 -9266.534,E2 -9266.534} C_VEL
LIN {X 0,Y 443.905,Z 335.973,A -85,B 0,C 180,E1 -9266.645,E2 -9266.645} C_VEL
LIN {X 0,Y 443.206,Z 341.817,A -85,B 0,C 180,E1 -9266.716,E2 -9266.716} C_VEL
LIN {X 0,Y 437.426,Z 360.794,A -85,B 0,C 180,E1 -9266.826,E2 -9266.826} C_VEL
LIN {X 0,Y 436.75,Z 366.638,A -85,B 0,C 180,E1 -9266.901,E2 -9266.901} C_VEL
LIN {X 0,Y 436.168,Z 419.655,A -85,B 0,C 180,E1 -9267.796,E2 -9267.796} C_VEL
LIN {X 0,Y 435.809,Z 432.256,A -85,B 0,C 180,E1 -9268.181,E2 -9268.181} C_VEL
LIN {X 0,Y 435.402,Z 445.474,A -85,B 0,C 180,E1 -9268.787,E2 -9268.787} C_VEL
LIN {X 0,Y 434.845,Z 457.421,A -85,B 0,C 180,E1 -9269.538,E2 -9269.538} C_VEL
LIN {X 0,Y 434.218,Z 468.836,A -85,B 0,C 180,E1 -9270.464,E2 -9270.464} C_VEL
LIN {X 0,Y 433.566,Z 479.141,A -85,B 0,C 180,E1 -9271.51,E2 -9271.51} C_VEL
LIN {X 0,Y 433.059,Z 487.555,A -85,B 0,C 180,E1 -9272.559,E2 -9272.559} C_VEL
LIN {X 0,Y 432.457,Z 496.691,A -85,B 0,C 180,E1 -9273.961,E2 -9273.961} C_VEL
LIN {X 0,Y 431.995,Z 504.053,A -85,B 0,C 180,E1 -9275.368,E2 -9275.368} C_VEL
LIN {X 0,Y 431.765,Z 510.109,A -85,B 0,C 180,E1 -9276.82,E2 -9276.82} C_VEL
LIN {X 0,Y 431.497,Z 515.281,A -85,B 0,C 180,E1 -9278.43,E2 -9278.43} C_VEL
LIN {X 0,Y 431.36,Z 517.649,A -85,B 0,C 180,E1 -9279.377,E2 -9279.377} C_VEL
LIN {X 0,Y 431.28,Z 519.583,A -85,B 0,C 180,E1 -9280.327,E2 -9280.327} C_VEL
LIN {X 0,Y 431.197,Z 521.964,A -85,B 0,C 180,E1 -9282.059,E2 -9282.059} C_VEL
LIN {X 0,Y 431.103,Z 522.765,A -85,B 0,C 180,E1 -9283.194,E2 -9283.194} C_VEL
LIN {X 0,Y 431.086,Z 523.016,A -85,B 0,C 180,E1 -9284.155,E2 -9284.155} C_VEL
LIN {X 0,Y 431.16,Z 522.346,A -85,B 0,C 180,E1 -9285.905,E2 -9285.905} C_VEL
LIN {X 0,Y 431.169,Z 521.164,A -85,B 0,C 180,E1 -9287.062,E2 -9287.062} C_VEL
LIN {X 0,Y 431.28,Z 519.679,A -85,B 0,C 180,E1 -9288.037,E2 -9288.037} C_VEL
LIN {X 0,Y 431.522,Z 516.693,A -85,B 0,C 180,E1 -9289.455,E2 -9289.455} C_VEL
LIN {X 0,Y 431.771,Z 512.284,A -85,B 0,C 180,E1 -9290.984,E2 -9290.984} C_VEL
LIN {X 0,Y 432.116,Z 506.694,A -85,B 0,C 180,E1 -9292.471,E2 -9292.471} C_VEL
LIN {X 0,Y 432.652,Z 499.606,A -85,B 0,C 180,E1 -9293.96,E2 -9293.96} C_VEL
LIN {X 0,Y 433.164,Z 492.268,A -85,B 0,C 180,E1 -9295.208,E2 -9295.208} C_VEL
LIN {X 0,Y 433.819,Z 483.26,A -85,B 0,C 180,E1 -9296.456,E2 -9296.456} C_VEL
LIN {X 0,Y 434.52,Z 473.202,A -85,B 0,C 180,E1 -9297.582,E2 -9297.582} C_VEL
LIN {X 0,Y 435.155,Z 463.635,A -85,B 0,C 180,E1 -9298.454,E2 -9298.454} C_VEL
LIN {X 0,Y 435.871,Z 451.473,A -85,B 0,C 180,E1 -9299.336,E2 -9299.336} C_VEL
LIN {X 0,Y 436.392,Z 438.906,A -85,B 0,C 180,E1 -9300.017,E2 -9300.017} C_VEL
LIN {X 0,Y 436.818,Z 425.759,A -85,B 0,C 180,E1 -9300.519,E2 -9300.519} C_VEL
LIN {X 0,Y 437.029,Z 411.867,A -85,B 0,C 180,E1 -9300.837,E2 -9300.837} C_VEL
LIN {X 0,Y 437.999,Z 330.271,A -85,B 0,C 180,E1 -9302.197,E2 -9302.197} C_VEL
LIN {X 0,Y 434.068,Z 312.211,A -85,B 0,C 180,E1 -9302.712,E2 -9302.712} C_VEL
LIN {X 0,Y 434.215,Z 306.24,A -85,B 0,C 180,E1 -9303.946,E2 -9303.946} C_VEL
LIN {X 0,Y 432.713,Z 298.418,A -85,B 0,C 180,E1 -9305.699,E2 -9305.699} C_VEL
LIN {X 0,Y 432.342,Z 296.633,A -85,B 0,C 180,E1 -9306.141,E2 -9306.141} C_VEL
LIN {X 0,Y 432.33,Z 296.63,A -85,B 0,C 180,E1 -9309.345,E2 -9309.345} C_VEL
LIN {X 0,Y 432.335,Z 296.631,A -85,B 0,C 180,E1 -9311.797,E2 -9311.797} C_VEL
LIN {X 0,Y 432.336,Z 296.635,A -85,B 0,C 180,E1 -9314.347,E2 -9314.347} C_VEL
LIN {X 0,Y 432.322,Z 296.632,A -85,B 0,C 180,E1 -9317.016,E2 -9317.016} C_VEL
LIN {X 0,Y 432.343,Z 296.628,A -85,B 0,C 180,E1 -9319.819,E2 -9319.819} C_VEL
LIN {X 0,Y 432.308,Z 296.637,A -85,B 0,C 180,E1 -9323.022,E2 -9323.022} C_VEL
LIN {X 0,Y 432.36,Z 296.626,A -85,B 0,C 180,E1 -9325.996,E2 -9325.996} C_VEL
LIN {X 0,Y 432.348,Z 296.625,A -85,B 0,C 180,E1 -9329.49,E2 -9329.49} C_VEL
LIN {X 0,Y 432.392,Z 296.624,A -85,B 0,C 180,E1 -9332.928,E2 -9332.928} C_VEL
LIN {X 0,Y 432.372,Z 296.622,A -85,B 0,C 180,E1 -9336.023,E2 -9336.023} C_VEL
LIN {X 0,Y 432.351,Z 296.629,A -85,B 0,C 180,E1 -9339.046,E2 -9339.046} C_VEL
LIN {X 0,Y 432.378,Z 296.622,A -85,B 0,C 180,E1 -9342.011,E2 -9342.011} C_VEL
LIN {X 0,Y 432.395,Z 296.62,A -85,B 0,C 180,E1 -9344.926,E2 -9344.926} C_VEL
LIN {X 0,Y 432.459,Z 296.617,A -85,B 0,C 180,E1 -9347.803,E2 -9347.803} C_VEL
LIN {X 0,Y 432.492,Z 296.607,A -85,B 0,C 180,E1 -9351.59,E2 -9351.59} C_VEL
LIN {X 0,Y 432.593,Z 296.593,A -85,B 0,C 180,E1 -9354.406,E2 -9354.406} C_VEL
LIN {X 0,Y 432.603,Z 296.598,A -85,B 0,C 180,E1 -9358.138,E2 -9358.138} C_VEL
LIN {X 0,Y 432.732,Z 296.577,A -85,B 0,C 180,E1 -9360,E2 -9360} C_VEL
LIN {X 0,Y 432.592,Z 296.594,A -85,B 0,C 180,E1 -9362.794,E2 -9362.794} C_VEL
LIN {X 0,Y 432.568,Z 296.597,A -85,B 0,C 180,E1 -9366.53,E2 -9366.53} C_VEL
LIN {X 0,Y 432.441,Z 296.612,A -85,B 0,C 180,E1 -9369.353,E2 -9369.353} C_VEL
LIN {X 0,Y 432.431,Z 296.617,A -85,B 0,C 180,E1 -9372.803,E2 -9372.803} C_VEL
LIN {X 0,Y 432.413,Z 296.617,A -85,B 0,C 180,E1 -9376.479,E2 -9376.479} C_VEL
LIN {X 0,Y 432.339,Z 296.627,A -85,B 0,C 180,E1 -9379.96,E2 -9379.96} C_VEL
LIN {X 0,Y 432.319,Z 296.634,A -85,B 0,C 180,E1 -9382.964,E2 -9382.964} C_VEL
LIN {X 0,Y 432.362,Z 296.618,A -85,B 0,C 180,E1 -9386.033,E2 -9386.033} C_VEL
LIN {X 0,Y 432.343,Z 296.625,A -85,B 0,C 180,E1 -9389.187,E2 -9389.187} C_VEL
LIN {X 0,Y 432.323,Z 296.631,A -85,B 0,C 180,E1 -9392.443,E2 -9392.443} C_VEL
LIN {X 0,Y 432.344,Z 296.628,A -85,B 0,C 180,E1 -9395.632,E2 -9395.632} C_VEL
LIN {X 0,Y 432.341,Z 296.628,A -85,B 0,C 180,E1 -9398.714,E2 -9398.714} C_VEL
LIN {X 0,Y 432.335,Z 296.631,A -85,B 0,C 180,E1 -9401.797,E2 -9401.797} C_VEL
LIN {X 0,Y 432.335,Z 296.629,A -85,B 0,C 180,E1 -9404.347,E2 -9404.347} C_VEL
LIN {X 0,Y 432.322,Z 296.632,A -85,B 0,C 180,E1 -9407.016,E2 -9407.016} C_VEL
LIN {X 0,Y 432.335,Z 296.628,A -85,B 0,C 180,E1 -9409.821,E2 -9409.821} C_VEL
LIN {X 0,Y 432.308,Z 296.635,A -85,B 0,C 180,E1 -9413.022,E2 -9413.022} C_VEL
LIN {X 0,Y 432.362,Z 296.628,A -85,B 0,C 180,E1 -9415.996,E2 -9415.996} C_VEL
LIN {X 0,Y 432.35,Z 296.628,A -85,B 0,C 180,E1 -9419.489,E2 -9419.489} C_VEL
LIN {X 0,Y 432.467,Z 296.823,A -85,B 0,C 180,E1 -9422.475,E2 -9422.475} C_VEL
LIN {X 0,Y 435.072,Z 309.485,A -85,B 0,C 180,E1 -9425.165,E2 -9425.165} C_VEL
LIN {X 0,Y 435.447,Z 313.392,A -85,B 0,C 180,E1 -9425.95,E2 -9425.95} C_VEL
LIN {X 0,Y 434.411,Z 329.006,A -85,B 0,C 180,E1 -9428.902,E2 -9428.902} C_VEL
LIN {X 0,Y 433.713,Z 341.892,A -85,B 0,C 180,E1 -9431.31,E2 -9431.31} C_VEL
LIN {X 0,Y 437.67,Z 366.066,A -85,B 0,C 180,E1 -9431.933,E2 -9431.933} C_VEL
LIN {X 0,Y 436.791,Z 450.837,A -85,B 0,C 180,E1 -9433.375,E2 -9433.375} C_VEL
LIN {X 0,Y 436.323,Z 463.909,A -85,B 0,C 180,E1 -9433.777,E2 -9433.777} C_VEL
LIN {X 0,Y 435.706,Z 475.97,A -85,B 0,C 180,E1 -9434.325,E2 -9434.325} C_VEL
LIN {X 0,Y 435.055,Z 487.366,A -85,B 0,C 180,E1 -9435.02,E2 -9435.02} C_VEL
LIN {X 0,Y 434.279,Z 499.093,A -85,B 0,C 180,E1 -9435.951,E2 -9435.951} C_VEL
LIN {X 0,Y 433.607,Z 509.627,A -85,B 0,C 180,E1 -9437.003,E2 -9437.003} C_VEL
LIN {X 0,Y 433.031,Z 518.254,A -85,B 0,C 180,E1 -9438.057,E2 -9438.057} C_VEL
LIN {X 0,Y 432.384,Z 526.224,A -85,B 0,C 180,E1 -9439.226,E2 -9439.226} C_VEL
LIN {X 0,Y 431.921,Z 534.055,A -85,B 0,C 180,E1 -9440.635,E2 -9440.635} C_VEL
LIN {X 0,Y 431.577,Z 540.332,A -85,B 0,C 180,E1 -9442.043,E2 -9442.043} C_VEL
LIN {X 0,Y 431.327,Z 546.055,A -85,B 0,C 180,E1 -9443.685,E2 -9443.685} C_VEL
LIN {X 0,Y 431.271,Z 550.296,A -85,B 0,C 180,E1 -9445.326,E2 -9445.326} C_VEL
LIN {X 0,Y 431.188,Z 552.078,A -85,B 0,C 180,E1 -9446.261,E2 -9446.261} C_VEL
LIN {X 0,Y 431.236,Z 553.436,A -85,B 0,C 180,E1 -9447.197,E2 -9447.197} C_VEL
LIN {X 0,Y 431.218,Z 554.397,A -85,B 0,C 180,E1 -9448.131,E2 -9448.131} C_VEL
LIN {X 0,Y 431.171,Z 554.969,A -85,B 0,C 180,E1 -9449.065,E2 -9449.065} C_VEL
LIN {X 0,Y 431.193,Z 555.113,A -85,B 0,C 180,E1 -9449.999,E2 -9449.999} C_VEL
LIN {X 0,Y 431.219,Z 554.206,A -85,B 0,C 180,E1 -9451.867,E2 -9451.867} C_VEL
LIN {X 0,Y 431.268,Z 553.169,A -85,B 0,C 180,E1 -9452.802,E2 -9452.802} C_VEL
LIN {X 0,Y 431.191,Z 551.68,A -85,B 0,C 180,E1 -9453.737,E2 -9453.737} C_VEL
LIN {X 0,Y 431.293,Z 548.651,A -85,B 0,C 180,E1 -9455.141,E2 -9455.141} C_VEL
LIN {X 0,Y 431.375,Z 544.552,A -85,B 0,C 180,E1 -9456.548,E2 -9456.548} C_VEL
LIN {X 0,Y 431.601,Z 538.255,A -85,B 0,C 180,E1 -9458.191,E2 -9458.191} C_VEL
LIN {X 0,Y 431.915,Z 531.393,A -85,B 0,C 180,E1 -9459.6,E2 -9459.6} C_VEL
LIN {X 0,Y 432.415,Z 522.837,A -85,B 0,C 180,E1 -9461.009,E2 -9461.009} C_VEL
LIN {X 0,Y 432.967,Z 514.028,A -85,B 0,C 180,E1 -9462.181,E2 -9462.181} C_VEL
LIN {X 0,Y 433.594,Z 503.723,A -85,B 0,C 180,E1 -9463.299,E2 -9463.299} C_VEL
LIN {X 0,Y 434.19,Z 492.314,A -85,B 0,C 180,E1 -9464.29,E2 -9464.29} C_VEL
LIN {X 0,Y 434.846,Z 480.11,A -85,B 0,C 180,E1 -9465.106,E2 -9465.106} C_VEL
LIN {X 0,Y 435.465,Z 467.351,A -85,B 0,C 180,E1 -9465.743,E2 -9465.743} C_VEL
LIN {X 0,Y 435.931,Z 454.702,A -85,B 0,C 180,E1 -9466.176,E2 -9466.176} C_VEL
LIN {X 0,Y 436.185,Z 438.556,A -85,B 0,C 180,E1 -9466.497,E2 -9466.497} C_VEL
LIN {X 0,Y 436.763,Z 365.498,A -85,B 0,C 180,E1 -9467.703,E2 -9467.703} C_VEL
LIN {X 0,Y 433.335,Z 342.33,A -85,B 0,C 180,E1 -9468.221,E2 -9468.221} C_VEL
LIN {X 0,Y 434.286,Z 324.012,A -85,B 0,C 180,E1 -9471.601,E2 -9471.601} C_VEL
LIN {X 0,Y 434.959,Z 310.74,A -85,B 0,C 180,E1 -9474.077,E2 -9474.077} C_VEL
LIN {X 0,Y 433.344,Z 301.247,A -85,B 0,C 180,E1 -9475.968,E2 -9475.968} C_VEL
LIN {X 0,Y 432.448,Z 296.618,A -85,B 0,C 180,E1 -9476.939,E2 -9476.939} C_VEL
LIN {X 0,Y 432.345,Z 296.632,A -85,B 0,C 180,E1 -9480.509,E2 -9480.509} C_VEL
LIN {X 0,Y 432.357,Z 296.629,A -85,B 0,C 180,E1 -9484.003,E2 -9484.003} C_VEL
LIN {X 0,Y 432.318,Z 296.629,A -85,B 0,C 180,E1 -9487.196,E2 -9487.196} C_VEL
LIN {X 0,Y 432.32,Z 296.634,A -85,B 0,C 180,E1 -9490.56,E2 -9490.56} C_VEL
LIN {X 0,Y 432.312,Z 296.63,A -85,B 0,C 180,E1 -9493.06,E2 -9493.06} C_VEL
LIN {X 0,Y 432.335,Z 296.627,A -85,B 0,C 180,E1 -9495.663,E2 -9495.663} C_VEL
LIN {X 0,Y 432.328,Z 296.633,A -85,B 0,C 180,E1 -9498.397,E2 -9498.397} C_VEL
LIN {X 0,Y 432.341,Z 296.626,A -85,B 0,C 180,E1 -9501.85,E2 -9501.85} C_VEL
LIN {X 0,Y 432.333,Z 296.628,A -85,B 0,C 180,E1 -9505.322,E2 -9505.322} C_VEL
LIN {X 0,Y 432.327,Z 296.633,A -85,B 0,C 180,E1 -9508.654,E2 -9508.654} C_VEL
LIN {X 0,Y 432.376,Z 296.621,A -85,B 0,C 180,E1 -9511.876,E2 -9511.876} C_VEL
LIN {X 0,Y 432.343,Z 296.634,A -85,B 0,C 180,E1 -9514.998,E2 -9514.998} C_VEL
LIN {X 0,Y 432.348,Z 296.625,A -85,B 0,C 180,E1 -9518.045,E2 -9518.045} C_VEL
LIN {X 0,Y 432.377,Z 296.628,A -85,B 0,C 180,E1 -9521.029,E2 -9521.029} C_VEL
LIN {X 0,Y 432.422,Z 296.616,A -85,B 0,C 180,E1 -9523.961,E2 -9523.961} C_VEL
LIN {X 0,Y 432.45,Z 296.615,A -85,B 0,C 180,E1 -9527.803,E2 -9527.803} C_VEL
LIN {X 0,Y 432.483,Z 296.615,A -85,B 0,C 180,E1 -9531.59,E2 -9531.59} C_VEL
LIN {X 0,Y 432.587,Z 296.595,A -85,B 0,C 180,E1 -9534.406,E2 -9534.406} C_VEL
LIN {X 0,Y 432.595,Z 296.596,A -85,B 0,C 180,E1 -9538.138,E2 -9538.138} C_VEL
LIN {X 0,Y 432.723,Z 296.582,A -85,B 0,C 180,E1 -9540,E2 -9540} C_VEL
LIN {X 0,Y 432.596,Z 296.594,A -85,B 0,C 180,E1 -9542.794,E2 -9542.794} C_VEL
LIN {X 0,Y 432.532,Z 296.603,A -85,B 0,C 180,E1 -9546.524,E2 -9546.524} C_VEL
LIN {X 0,Y 432.433,Z 296.616,A -85,B 0,C 180,E1 -9549.353,E2 -9549.353} C_VEL
LIN {X 0,Y 432.421,Z 296.616,A -85,B 0,C 180,E1 -9552.804,E2 -9552.804} C_VEL
LIN {X 0,Y 432.414,Z 296.62,A -85,B 0,C 180,E1 -9556.484,E2 -9556.484} C_VEL
LIN {X 0,Y 432.33,Z 296.632,A -85,B 0,C 180,E1 -9559.961,E2 -9559.961} C_VEL
LIN {X 0,Y 432.308,Z 296.631,A -85,B 0,C 180,E1 -9562.965,E2 -9562.965} C_VEL
LIN {X 0,Y 432.342,Z 296.629,A -85,B 0,C 180,E1 -9566.034,E2 -9566.034} C_VEL
LIN {X 0,Y 432.334,Z 296.627,A -85,B 0,C 180,E1 -9569.188,E2 -9569.188} C_VEL
LIN {X 0,Y 432.315,Z 296.636,A -85,B 0,C 180,E1 -9572.444,E2 -9572.444} C_VEL
LIN {X 0,Y 432.337,Z 296.626,A -85,B 0,C 180,E1 -9575.633,E2 -9575.633} C_VEL
LIN {X 0,Y 432.319,Z 296.637,A -85,B 0,C 180,E1 -9578.713,E2 -9578.713} C_VEL
LIN {X 0,Y 432.314,Z 296.629,A -85,B 0,C 180,E1 -9581.8,E2 -9581.8} C_VEL
LIN {X 0,Y 432.328,Z 296.629,A -85,B 0,C 180,E1 -9584.348,E2 -9584.348} C_VEL
LIN {X 0,Y 432.301,Z 296.638,A -85,B 0,C 180,E1 -9587.019,E2 -9587.019} C_VEL
LIN {X 0,Y 432.304,Z 296.631,A -85,B 0,C 180,E1 -9589.826,E2 -9589.826} C_VEL
LIN {X 0,Y 432.3,Z 296.638,A -85,B 0,C 180,E1 -9593.023,E2 -9593.023} C_VEL
LIN {X 0,Y 432.354,Z 296.624,A -85,B 0,C 180,E1 -9595.998,E2 -9595.998} C_VEL
LIN {X 0,Y 432.341,Z 296.631,A -85,B 0,C 180,E1 -9599.492,E2 -9599.492} C_VEL
LIN {X 0,Y 432.317,Z 296.63,A -85,B 0,C 180,E1 -9601.873,E2 -9601.873} C_VEL
LIN {X 0,Y 432.32,Z 296.631,A -85,B 0,C 180,E1 -9604.998,E2 -9604.998} C_VEL
LIN {X 0,Y 432.357,Z 296.625,A -85,B 0,C 180,E1 -9608.047,E2 -9608.047} C_VEL
LIN {X 0,Y 432.384,Z 296.622,A -85,B 0,C 180,E1 -9611.03,E2 -9611.03} C_VEL
LIN {X 0,Y 432.429,Z 296.619,A -85,B 0,C 180,E1 -9613.962,E2 -9613.962} C_VEL
LIN {X 0,Y 432.451,Z 296.62,A -85,B 0,C 180,E1 -9617.804,E2 -9617.804} C_VEL
LIN {X 0,Y 432.446,Z 296.621,A -85,B 0,C 180,E1 -9621.59,E2 -9621.59} C_VEL
LIN {X 0,Y 432.537,Z 296.787,A -85,B 0,C 180,E1 -9622.532,E2 -9622.532} C_VEL
LIN {X 0,Y 433.745,Z 304.203,A -85,B 0,C 180,E1 -9624.189,E2 -9624.189} C_VEL
LIN {X 0,Y 433.603,Z 312.317,A -85,B 0,C 180,E1 -9625.865,E2 -9625.865} C_VEL
LIN {X 0,Y 437.099,Z 330.999,A -85,B 0,C 180,E1 -9626.313,E2 -9626.313} C_VEL
LIN {X 0,Y 436.75,Z 366.638,A -85,B 0,C 180,E1 -9626.901,E2 -9626.901} C_VEL
LIN {X 0,Y 436.082,Z 372.479,A -85,B 0,C 180,E1 -9626.975,E2 -9626.975} C_VEL
LIN {X 0,Y 430.312,Z 391.45,A -85,B 0,C 180,E1 -9627.093,E2 -9627.093} C_VEL
LIN {X 0,Y 429.567,Z 397.294,A -85,B 0,C 180,E1 -9627.166,E2 -9627.166} C_VEL
LIN {X 0,Y 429.26,Z 421.163,A -85,B 0,C 180,E1 -9627.601,E2 -9627.601} C_VEL
LIN {X 0,Y 428.858,Z 434.723,A -85,B 0,C 180,E1 -9628.045,E2 -9628.045} C_VEL
LIN {X 0,Y 428.443,Z 447.051,A -85,B 0,C 180,E1 -9628.65,E2 -9628.65} C_VEL
LIN {X 0,Y 427.866,Z 458.687,A -85,B 0,C 180,E1 -9629.412,E2 -9629.412} C_VEL
LIN {X 0,Y 427.212,Z 469.92,A -85,B 0,C 180,E1 -9630.354,E2 -9630.354} C_VEL
LIN {X 0,Y 426.558,Z 480.058,A -85,B 0,C 180,E1 -9631.417,E2 -9631.417} C_VEL
LIN {X 0,Y 425.958,Z 489.179,A -85,B 0,C 180,E1 -9632.601,E2 -9632.601} C_VEL
LIN {X 0,Y 425.36,Z 498.074,A -85,B 0,C 180,E1 -9634.027,E2 -9634.027} C_VEL
LIN {X 0,Y 424.896,Z 505.24,A -85,B 0,C 180,E1 -9635.458,E2 -9635.458} C_VEL
LIN {X 0,Y 424.686,Z 510.686,A -85,B 0,C 180,E1 -9636.819,E2 -9636.819} C_VEL
LIN {X 0,Y 424.467,Z 514.767,A -85,B 0,C 180,E1 -9638.091,E2 -9638.091} C_VEL
LIN {X 0,Y 424.247,Z 518.367,A -85,B 0,C 180,E1 -9639.536,E2 -9639.536} C_VEL
LIN {X 0,Y 424.171,Z 520.202,A -85,B 0,C 180,E1 -9640.502,E2 -9640.502} C_VEL
LIN {X 0,Y 424.106,Z 522.279,A -85,B 0,C 180,E1 -9642.119,E2 -9642.119} C_VEL
LIN {X 0,Y 423.995,Z 523.134,A -85,B 0,C 180,E1 -9643.419,E2 -9643.419} C_VEL
LIN {X 0,Y 423.991,Z 523.262,A -85,B 0,C 180,E1 -9644.397,E2 -9644.397} C_VEL
LIN {X 0,Y 424.091,Z 522.572,A -85,B 0,C 180,E1 -9646.018,E2 -9646.018} C_VEL
LIN {X 0,Y 424.103,Z 521.163,A -85,B 0,C 180,E1 -9647.355,E2 -9647.355} C_VEL
LIN {X 0,Y 424.234,Z 519.56,A -85,B 0,C 180,E1 -9648.347,E2 -9648.347} C_VEL
LIN {X 0,Y 424.515,Z 516.295,A -85,B 0,C 180,E1 -9649.84,E2 -9649.84} C_VEL
LIN {X 0,Y 424.795,Z 511.853,A -85,B 0,C 180,E1 -9651.345,E2 -9651.345} C_VEL
LIN {X 0,Y 425.185,Z 506.09,A -85,B 0,C 180,E1 -9652.858,E2 -9652.858} C_VEL
LIN {X 0,Y 425.781,Z 498.766,A -85,B 0,C 180,E1 -9654.372,E2 -9654.372} C_VEL
LIN {X 0,Y 426.361,Z 491.16,A -85,B 0,C 180,E1 -9655.639,E2 -9655.639} C_VEL
LIN {X 0,Y 427.047,Z 481.817,A -85,B 0,C 180,E1 -9656.909,E2 -9656.909} C_VEL
LIN {X 0,Y 427.804,Z 471.423,A -85,B 0,C 180,E1 -9658.051,E2 -9658.051} C_VEL
LIN {X 0,Y 428.578,Z 461.392,A -85,B 0,C 180,E1 -9658.931,E2 -9658.931} C_VEL
LIN {X 0,Y 429.226,Z 448.898,A -85,B 0,C 180,E1 -9659.795,E2 -9659.795} C_VEL
LIN {X 0,Y 429.766,Z 435.956,A -85,B 0,C 180,E1 -9660.461,E2 -9660.461} C_VEL
LIN {X 0,Y 430.208,Z 423.187,A -85,B 0,C 180,E1 -9660.902,E2 -9660.902} C_VEL
LIN {X 0,Y 430.448,Z 407.317,A -85,B 0,C 180,E1 -9661.224,E2 -9661.224} C_VEL
LIN {X 0,Y 431.349,Z 330.972,A -85,B 0,C 180,E1 -9662.523,E2 -9662.523} C_VEL
LIN {X 0,Y 427.2,Z 312.334,A -85,B 0,C 180,E1 -9663.088,E2 -9663.088} C_VEL
LIN {X 0,Y 427.222,Z 306.642,A -85,B 0,C 180,E1 -9664.301,E2 -9664.301} C_VEL
LIN {X 0,Y 425.299,Z 297.511,A -85,B 0,C 180,E1 -9666.42,E2 -9666.42} C_VEL
LIN {X 0,Y 425.284,Z 297.508,A -85,B 0,C 180,E1 -9669.041,E2 -9669.041} C_VEL
LIN {X 0,Y 425.292,Z 297.509,A -85,B 0,C 180,E1 -9671.958,E2 -9671.958} C_VEL
LIN {X 0,Y 425.287,Z 297.51,A -85,B 0,C 180,E1 -9675.283,E2 -9675.283} C_VEL
LIN {X 0,Y 425.278,Z 297.518,A -85,B 0,C 180,E1 -9678.621,E2 -9678.621} C_VEL
LIN {X 0,Y 425.314,Z 297.501,A -85,B 0,C 180,E1 -9681.103,E2 -9681.103} C_VEL
LIN {X 0,Y 425.3,Z 297.508,A -85,B 0,C 180,E1 -9684.664,E2 -9684.664} C_VEL
LIN {X 0,Y 425.266,Z 297.509,A -85,B 0,C 180,E1 -9688.073,E2 -9688.073} C_VEL
LIN {X 0,Y 425.332,Z 297.504,A -85,B 0,C 180,E1 -9691.368,E2 -9691.368} C_VEL
LIN {X 0,Y 425.296,Z 297.505,A -85,B 0,C 180,E1 -9694.555,E2 -9694.555} C_VEL
LIN {X 0,Y 425.289,Z 297.508,A -85,B 0,C 180,E1 -9697.661,E2 -9697.661} C_VEL
LIN {X 0,Y 425.363,Z 297.494,A -85,B 0,C 180,E1 -9700.704,E2 -9700.704} C_VEL
LIN {X 0,Y 425.389,Z 297.496,A -85,B 0,C 180,E1 -9703.688,E2 -9703.688} C_VEL
LIN {X 0,Y 425.412,Z 297.496,A -85,B 0,C 180,E1 -9707.598,E2 -9707.598} C_VEL
LIN {X 0,Y 425.443,Z 297.483,A -85,B 0,C 180,E1 -9711.45,E2 -9711.45} C_VEL
LIN {X 0,Y 425.55,Z 297.471,A -85,B 0,C 180,E1 -9714.313,E2 -9714.313} C_VEL
LIN {X 0,Y 425.573,Z 297.474,A -85,B 0,C 180,E1 -9718.107,E2 -9718.107} C_VEL
LIN {X 0,Y 425.701,Z 297.452,A -85,B 0,C 180,E1 -9720,E2 -9720} C_VEL
LIN {X 0,Y 425.546,Z 297.472,A -85,B 0,C 180,E1 -9722.84,E2 -9722.84} C_VEL
LIN {X 0,Y 425.527,Z 297.473,A -85,B 0,C 180,E1 -9726.639,E2 -9726.639} C_VEL
LIN {X 0,Y 425.4,Z 297.49,A -85,B 0,C 180,E1 -9729.509,E2 -9729.509} C_VEL
LIN {X 0,Y 425.394,Z 297.493,A -85,B 0,C 180,E1 -9732.904,E2 -9732.904} C_VEL
LIN {X 0,Y 425.362,Z 297.495,A -85,B 0,C 180,E1 -9736.605,E2 -9736.605} C_VEL
LIN {X 0,Y 425.329,Z 297.499,A -85,B 0,C 180,E1 -9739.636,E2 -9739.636} C_VEL
LIN {X 0,Y 425.288,Z 297.505,A -85,B 0,C 180,E1 -9742.339,E2 -9742.339} C_VEL
LIN {X 0,Y 425.293,Z 297.499,A -85,B 0,C 180,E1 -9745.446,E2 -9745.446} C_VEL
LIN {X 0,Y 425.332,Z 297.505,A -85,B 0,C 180,E1 -9748.632,E2 -9748.632} C_VEL
LIN {X 0,Y 425.265,Z 297.508,A -85,B 0,C 180,E1 -9751.927,E2 -9751.927} C_VEL
LIN {X 0,Y 425.298,Z 297.509,A -85,B 0,C 180,E1 -9755.336,E2 -9755.336} C_VEL
LIN {X 0,Y 425.303,Z 297.507,A -85,B 0,C 180,E1 -9758.898,E2 -9758.898} C_VEL
LIN {X 0,Y 425.291,Z 297.507,A -85,B 0,C 180,E1 -9761.958,E2 -9761.958} C_VEL
LIN {X 0,Y 425.286,Z 297.512,A -85,B 0,C 180,E1 -9765.283,E2 -9765.283} C_VEL
LIN {X 0,Y 425.276,Z 297.508,A -85,B 0,C 180,E1 -9768.621,E2 -9768.621} C_VEL
LIN {X 0,Y 425.299,Z 297.501,A -85,B 0,C 180,E1 -9771.101,E2 -9771.101} C_VEL
LIN {X 0,Y 425.302,Z 297.505,A -85,B 0,C 180,E1 -9774.664,E2 -9774.664} C_VEL
LIN {X 0,Y 425.268,Z 297.513,A -85,B 0,C 180,E1 -9778.073,E2 -9778.073} C_VEL
LIN {X 0,Y 425.334,Z 297.505,A -85,B 0,C 180,E1 -9781.368,E2 -9781.368} C_VEL
LIN {X 0,Y 425.378,Z 297.632,A -85,B 0,C 180,E1 -9782.143,E2 -9782.143} C_VEL
LIN {X 0,Y 427.913,Z 309.475,A -85,B 0,C 180,E1 -9784.721,E2 -9784.721} C_VEL
LIN {X 0,Y 428.556,Z 314.667,A -85,B 0,C 180,E1 -9785.796,E2 -9785.796} C_VEL
LIN {X 0,Y 427.359,Z 332.879,A -85,B 0,C 180,E1 -9789.294,E2 -9789.294} C_VEL
LIN {X 0,Y 426.811,Z 341.621,A -85,B 0,C 180,E1 -9790.953,E2 -9790.953} C_VEL
LIN {X 0,Y 430.623,Z 364.222,A -85,B 0,C 180,E1 -9791.556,E2 -9791.556} C_VEL
LIN {X 0,Y 431.033,Z 369.473,A -85,B 0,C 180,E1 -9791.669,E2 -9791.669} C_VEL
LIN {X 0,Y 430.083,Z 450.87,A -85,B 0,C 180,E1 -9793.077,E2 -9793.077} C_VEL
LIN {X 0,Y 429.58,Z 463.842,A -85,B 0,C 180,E1 -9793.485,E2 -9793.485} C_VEL
LIN {X 0,Y 428.909,Z 476.412,A -85,B 0,C 180,E1 -9794.07,E2 -9794.07} C_VEL
LIN {X 0,Y 428.221,Z 487.618,A -85,B 0,C 180,E1 -9794.776,E2 -9794.776} C_VEL
LIN {X 0,Y 427.395,Z 499.232,A -85,B 0,C 180,E1 -9795.72,E2 -9795.72} C_VEL
LIN {X 0,Y 426.669,Z 509.696,A -85,B 0,C 180,E1 -9796.788,E2 -9796.788} C_VEL
LIN {X 0,Y 426.07,Z 518.267,A -85,B 0,C 180,E1 -9797.859,E2 -9797.859} C_VEL
LIN {X 0,Y 425.398,Z 526.186,A -85,B 0,C 180,E1 -9799.047,E2 -9799.047} C_VEL
LIN {X 0,Y 424.872,Z 533.952,A -85,B 0,C 180,E1 -9800.478,E2 -9800.478} C_VEL
LIN {X 0,Y 424.523,Z 540.192,A -85,B 0,C 180,E1 -9801.91,E2 -9801.91} C_VEL
LIN {X 0,Y 424.301,Z 545.167,A -85,B 0,C 180,E1 -9803.341,E2 -9803.341} C_VEL
LIN {X 0,Y 424.206,Z 549.023,A -85,B 0,C 180,E1 -9804.771,E2 -9804.771} C_VEL
LIN {X 0,Y 424.1,Z 551.858,A -85,B 0,C 180,E1 -9806.199,E2 -9806.199} C_VEL
LIN {X 0,Y 424.133,Z 553.206,A -85,B 0,C 180,E1 -9807.15,E2 -9807.15} C_VEL
LIN {X 0,Y 424.143,Z 554.159,A -85,B 0,C 180,E1 -9808.1,E2 -9808.1} C_VEL
LIN {X 0,Y 424.091,Z 554.717,A -85,B 0,C 180,E1 -9809.05,E2 -9809.05} C_VEL
LIN {X 0,Y 424.108,Z 554.844,A -85,B 0,C 180,E1 -9809.999,E2 -9809.999} C_VEL
LIN {X 0,Y 424.145,Z 553.916,A -85,B 0,C 180,E1 -9811.898,E2 -9811.898} C_VEL
LIN {X 0,Y 424.163,Z 552.865,A -85,B 0,C 180,E1 -9812.848,E2 -9812.848} C_VEL
LIN {X 0,Y 424.102,Z 551.356,A -85,B 0,C 180,E1 -9813.8,E2 -9813.8} C_VEL
LIN {X 0,Y 424.206,Z 548.303,A -85,B 0,C 180,E1 -9815.227,E2 -9815.227} C_VEL
LIN {X 0,Y 424.299,Z 544.18,A -85,B 0,C 180,E1 -9816.657,E2 -9816.657} C_VEL
LIN {X 0,Y 424.534,Z 537.855,A -85,B 0,C 180,E1 -9818.328,E2 -9818.328} C_VEL
LIN {X 0,Y 424.883,Z 530.959,A -85,B 0,C 180,E1 -9819.761,E2 -9819.761} C_VEL
LIN {X 0,Y 425.282,Z 523.912,A -85,B 0,C 180,E1 -9820.954,E2 -9820.954} C_VEL
LIN {X 0,Y 425.881,Z 515.427,A -85,B 0,C 180,E1 -9822.145,E2 -9822.145} C_VEL
LIN {X 0,Y 426.549,Z 504.927,A -85,B 0,C 180,E1 -9823.336,E2 -9823.336} C_VEL
LIN {X 0,Y 427.13,Z 494.523,A -85,B 0,C 180,E1 -9824.288,E2 -9824.288} C_VEL
LIN {X 0,Y 427.744,Z 483.121,A -85,B 0,C 180,E1 -9825.119,E2 -9825.119} C_VEL
LIN {X 0,Y 428.375,Z 471.467,A -85,B 0,C 180,E1 -9825.766,E2 -9825.766} C_VEL
LIN {X 0,Y 428.892,Z 458.029,A -85,B 0,C 180,E1 -9826.296,E2 -9826.296} C_VEL
LIN {X 0,Y 429.236,Z 444.846,A -85,B 0,C 180,E1 -9826.619,E2 -9826.619} C_VEL
LIN {X 0,Y 429.98,Z 367.174,A -85,B 0,C 180,E1 -9827.919,E2 -9827.919} C_VEL
LIN {X 0,Y 426.352,Z 342.008,A -85,B 0,C 180,E1 -9828.5,E2 -9828.5} C_VEL
LIN {X 0,Y 427.31,Z 324.834,A -85,B 0,C 180,E1 -9831.718,E2 -9831.718} C_VEL
LIN {X 0,Y 427.986,Z 311.552,A -85,B 0,C 180,E1 -9834.237,E2 -9834.237} C_VEL
LIN {X 0,Y 425.996,Z 300.695,A -85,B 0,C 180,E1 -9836.45,E2 -9836.45} C_VEL
LIN {X 0,Y 425.401,Z 297.497,A -85,B 0,C 180,E1 -9837.165,E2 -9837.165} C_VEL
LIN {X 0,Y 425.285,Z 297.508,A -85,B 0,C 180,E1 -9840.815,E2 -9840.815} C_VEL
LIN {X 0,Y 425.309,Z 297.509,A -85,B 0,C 180,E1 -9844.287,E2 -9844.287} C_VEL
LIN {X 0,Y 425.274,Z 297.507,A -85,B 0,C 180,E1 -9847.693,E2 -9847.693} C_VEL
LIN {X 0,Y 425.275,Z 297.512,A -85,B 0,C 180,E1 -9850.519,E2 -9850.519} C_VEL
LIN {X 0,Y 425.252,Z 297.509,A -85,B 0,C 180,E1 -9853.35,E2 -9853.35} C_VEL
LIN {X 0,Y 425.259,Z 297.515,A -85,B 0,C 180,E1 -9856.647,E2 -9856.647} C_VEL
LIN {X 0,Y 425.288,Z 297.505,A -85,B 0,C 180,E1 -9859.873,E2 -9859.873} C_VEL
LIN {X 0,Y 425.278,Z 297.511,A -85,B 0,C 180,E1 -9862.486,E2 -9862.486} C_VEL
LIN {X 0,Y 425.3,Z 297.503,A -85,B 0,C 180,E1 -9865.817,E2 -9865.817} C_VEL
LIN {X 0,Y 425.298,Z 297.506,A -85,B 0,C 180,E1 -9869.235,E2 -9869.235} C_VEL
LIN {X 0,Y 425.343,Z 297.5,A -85,B 0,C 180,E1 -9872.442,E2 -9872.442} C_VEL
LIN {X 0,Y 425.343,Z 297.499,A -85,B 0,C 180,E1 -9875.602,E2 -9875.602} C_VEL
LIN {X 0,Y 425.284,Z 297.508,A -85,B 0,C 180,E1 -9878.681,E2 -9878.681} C_VEL
LIN {X 0,Y 425.324,Z 297.502,A -85,B 0,C 180,E1 -9881.702,E2 -9881.702} C_VEL
LIN {X 0,Y 425.34,Z 297.499,A -85,B 0,C 180,E1 -9884.67,E2 -9884.67} C_VEL
LIN {X 0,Y 425.403,Z 297.495,A -85,B 0,C 180,E1 -9887.598,E2 -9887.598} C_VEL
LIN {X 0,Y 425.433,Z 297.495,A -85,B 0,C 180,E1 -9891.45,E2 -9891.45} C_VEL
LIN {X 0,Y 425.544,Z 297.473,A -85,B 0,C 180,E1 -9894.313,E2 -9894.313} C_VEL
LIN {X 0,Y 425.565,Z 297.472,A -85,B 0,C 180,E1 -9898.107,E2 -9898.107} C_VEL
LIN {X 0,Y 425.693,Z 297.458,A -85,B 0,C 180,E1 -9900,E2 -9900} C_VEL
LIN {X 0,Y 425.548,Z 297.472,A -85,B 0,C 180,E1 -9902.84,E2 -9902.84} C_VEL
LIN {X 0,Y 425.487,Z 297.48,A -85,B 0,C 180,E1 -9906.524,E2 -9906.524} C_VEL
LIN {X 0,Y 425.391,Z 297.494,A -85,B 0,C 180,E1 -9909.51,E2 -9909.51} C_VEL
LIN {X 0,Y 425.384,Z 297.492,A -85,B 0,C 180,E1 -9912.904,E2 -9912.904} C_VEL
LIN {X 0,Y 425.361,Z 297.497,A -85,B 0,C 180,E1 -9916.609,E2 -9916.609} C_VEL
LIN {X 0,Y 425.32,Z 297.502,A -85,B 0,C 180,E1 -9919.636,E2 -9919.636} C_VEL
LIN {X 0,Y 425.279,Z 297.513,A -85,B 0,C 180,E1 -9922.339,E2 -9922.339} C_VEL
LIN {X 0,Y 425.312,Z 297.505,A -85,B 0,C 180,E1 -9924.658,E2 -9924.658} C_VEL
LIN {X 0,Y 425.337,Z 297.498,A -85,B 0,C 180,E1 -9927.559,E2 -9927.559} C_VEL
LIN {X 0,Y 425.28,Z 297.509,A -85,B 0,C 180,E1 -9930.817,E2 -9930.817} C_VEL
LIN {X 0,Y 425.304,Z 297.507,A -85,B 0,C 180,E1 -9934.289,E2 -9934.289} C_VEL
LIN {X 0,Y 425.269,Z 297.507,A -85,B 0,C 180,E1 -9937.696,E2 -9937.696} C_VEL
LIN {X 0,Y 425.24,Z 297.515,A -85,B 0,C 180,E1 -9940.516,E2 -9940.516} C_VEL
LIN {X 0,Y 425.249,Z 297.511,A -85,B 0,C 180,E1 -9943.351,E2 -9943.351} C_VEL
LIN {X 0,Y 425.252,Z 297.509,A -85,B 0,C 180,E1 -9946.045,E2 -9946.045} C_VEL
LIN {X 0,Y 425.25,Z 297.511,A -85,B 0,C 180,E1 -9949.485,E2 -9949.485} C_VEL
LIN {X 0,Y 425.272,Z 297.508,A -85,B 0,C 180,E1 -9952.49,E2 -9952.49} C_VEL
LIN {X 0,Y 425.302,Z 297.504,A -85,B 0,C 180,E1 -9955.818,E2 -9955.818} C_VEL
LIN {X 0,Y 425.287,Z 297.513,A -85,B 0,C 180,E1 -9959.24,E2 -9959.24} C_VEL
LIN {X 0,Y 425.244,Z 297.51,A -85,B 0,C 180,E1 -9962.436,E2 -9962.436} C_VEL
LIN {X 0,Y 425.318,Z 297.506,A -85,B 0,C 180,E1 -9965.601,E2 -9965.601} C_VEL
LIN {X 0,Y 425.292,Z 297.504,A -85,B 0,C 180,E1 -9968.683,E2 -9968.683} C_VEL
LIN {X 0,Y 425.32,Z 297.507,A -85,B 0,C 180,E1 -9971.703,E2 -9971.703} C_VEL
LIN {X 0,Y 425.344,Z 297.497,A -85,B 0,C 180,E1 -9974.671,E2 -9974.671} C_VEL
LIN {X 0,Y 425.407,Z 297.496,A -85,B 0,C 180,E1 -9977.599,E2 -9977.599} C_VEL
LIN {X 0,Y 425.394,Z 297.499,A -85,B 0,C 180,E1 -9981.45,E2 -9981.45} C_VEL
LIN {X 0,Y 425.481,Z 297.591,A -85,B 0,C 180,E1 -9982.337,E2 -9982.337} C_VEL
LIN {X 0,Y 426.769,Z 305.335,A -85,B 0,C 180,E1 -9984.093,E2 -9984.093} C_VEL
LIN {X 0,Y 426.603,Z 312.326,A -85,B 0,C 180,E1 -9985.59,E2 -9985.59} C_VEL
LIN {X 0,Y 430.246,Z 331.02,A -85,B 0,C 180,E1 -9986.057,E2 -9986.057} C_VEL
LIN {X 0,Y 429.567,Z 397.294,A -85,B 0,C 180,E1 -9987.166,E2 -9987.166} C_VEL
LIN {X 0,Y 428.826,Z 403.143,A -85,B 0,C 180,E1 -9987.237,E2 -9987.237} C_VEL
LIN {X 0,Y 422.943,Z 422.06,A -85,B 0,C 180,E1 -9987.401,E2 -9987.401} C_VEL
LIN {X 0,Y 422.186,Z 427.807,A -85,B 0,C 180,E1 -9987.552,E2 -9987.552} C_VEL
LIN {X 0,Y 421.772,Z 441.006,A -85,B 0,C 180,E1 -9988.091,E2 -9988.091} C_VEL
LIN {X 0,Y 421.21,Z 453.322,A -85,B 0,C 180,E1 -9988.806,E2 -9988.806} C_VEL
LIN {X 0,Y 420.653,Z 464.368,A -85,B 0,C 180,E1 -9989.642,E2 -9989.642} C_VEL
LIN {X 0,Y 420.03,Z 474.51,A -85,B 0,C 180,E1 -9990.6,E2 -9990.6} C_VEL
LIN {X 0,Y 419.323,Z 483.865,A -85,B 0,C 180,E1 -9991.681,E2 -9991.681} C_VEL
LIN {X 0,Y 418.737,Z 492.379,A -85,B 0,C 180,E1 -9992.887,E2 -9992.887} C_VEL
LIN {X 0,Y 418.225,Z 500.654,A -85,B 0,C 180,E1 -9994.337,E2 -9994.337} C_VEL
LIN {X 0,Y 417.785,Z 507.342,A -85,B 0,C 180,E1 -9995.793,E2 -9995.793} C_VEL
LIN {X 0,Y 417.528,Z 512.515,A -85,B 0,C 180,E1 -9997.205,E2 -9997.205} C_VEL
LIN {X 0,Y 417.285,Z 516.85,A -85,B 0,C 180,E1 -9998.719,E2 -9998.719} C_VEL
LIN {X 0,Y 417.133,Z 519.054,A -85,B 0,C 180,E1 -9999.7,E2 -9999.7} C_VEL
LIN {X 0,Y 417.076,Z 520.768,A -85,B 0,C 180,E1 -10000.683,E2 -10000.683} C_VEL
LIN {X 0,Y 417.015,Z 522.59,A -85,B 0,C 180,E1 -10002.181,E2 -10002.181} C_VEL
LIN {X 0,Y 416.916,Z 523.448,A -85,B 0,C 180,E1 -10003.651,E2 -10003.651} C_VEL
LIN {X 0,Y 416.912,Z 523.495,A -85,B 0,C 180,E1 -10004.647,E2 -10004.647} C_VEL
LIN {X 0,Y 417.014,Z 522.805,A -85,B 0,C 180,E1 -10006.13,E2 -10006.13} C_VEL
LIN {X 0,Y 417.051,Z 521.121,A -85,B 0,C 180,E1 -10007.658,E2 -10007.658} C_VEL
LIN {X 0,Y 417.349,Z 517.862,A -85,B 0,C 180,E1 -10009.434,E2 -10009.434} C_VEL
LIN {X 0,Y 417.691,Z 513.105,A -85,B 0,C 180,E1 -10011.208,E2 -10011.208} C_VEL
LIN {X 0,Y 418.113,Z 507.595,A -85,B 0,C 180,E1 -10012.744,E2 -10012.744} C_VEL
LIN {X 0,Y 418.714,Z 500.588,A -85,B 0,C 180,E1 -10014.282,E2 -10014.282} C_VEL
LIN {X 0,Y 419.299,Z 493.107,A -85,B 0,C 180,E1 -10015.61,E2 -10015.61} C_VEL
LIN {X 0,Y 419.986,Z 484.506,A -85,B 0,C 180,E1 -10016.861,E2 -10016.861} C_VEL
LIN {X 0,Y 420.799,Z 474.649,A -85,B 0,C 180,E1 -10018.017,E2 -10018.017} C_VEL
LIN {X 0,Y 421.648,Z 463.775,A -85,B 0,C 180,E1 -10019.043,E2 -10019.043} C_VEL
LIN {X 0,Y 422.366,Z 451.632,A -85,B 0,C 180,E1 -10019.947,E2 -10019.947} C_VEL
LIN {X 0,Y 422.948,Z 439.911,A -85,B 0,C 180,E1 -10020.601,E2 -10020.601} C_VEL
LIN {X 0,Y 423.404,Z 427.285,A -85,B 0,C 180,E1 -10021.107,E2 -10021.107} C_VEL
LIN {X 0,Y 423.68,Z 414.402,A -85,B 0,C 180,E1 -10021.432,E2 -10021.432} C_VEL
LIN {X 0,Y 424.798,Z 332.278,A -85,B 0,C 180,E1 -10022.846,E2 -10022.846} C_VEL
LIN {X 0,Y 420.684,Z 314.134,A -85,B 0,C 180,E1 -10023.4,E2 -10023.4} C_VEL
LIN {X 0,Y 420.378,Z 312.566,A -85,B 0,C 180,E1 -10023.463,E2 -10023.463} C_VEL
LIN {X 0,Y 420.387,Z 308.486,A -85,B 0,C 180,E1 -10024.349,E2 -10024.349} C_VEL
LIN {X 0,Y 418.233,Z 298.387,A -85,B 0,C 180,E1 -10026.77,E2 -10026.77} C_VEL
LIN {X 0,Y 418.247,Z 298.386,A -85,B 0,C 180,E1 -10029.683,E2 -10029.683} C_VEL
LIN {X 0,Y 418.232,Z 298.392,A -85,B 0,C 180,E1 -10032.321,E2 -10032.321} C_VEL
LIN {X 0,Y 418.238,Z 298.389,A -85,B 0,C 180,E1 -10035.109,E2 -10035.109} C_VEL
LIN {X 0,Y 418.242,Z 298.386,A -85,B 0,C 180,E1 -10037.767,E2 -10037.767} C_VEL
LIN {X 0,Y 418.26,Z 298.379,A -85,B 0,C 180,E1 -10040.618,E2 -10040.618} C_VEL
LIN {X 0,Y 418.244,Z 298.384,A -85,B 0,C 180,E1 -10043.976,E2 -10043.976} C_VEL
LIN {X 0,Y 418.259,Z 298.385,A -85,B 0,C 180,E1 -10047.156,E2 -10047.156} C_VEL
LIN {X 0,Y 418.27,Z 298.382,A -85,B 0,C 180,E1 -10050.895,E2 -10050.895} C_VEL
LIN {X 0,Y 418.271,Z 298.379,A -85,B 0,C 180,E1 -10054.096,E2 -10054.096} C_VEL
LIN {X 0,Y 418.239,Z 298.384,A -85,B 0,C 180,E1 -10057.264,E2 -10057.264} C_VEL
LIN {X 0,Y 418.284,Z 298.375,A -85,B 0,C 180,E1 -10060.364,E2 -10060.364} C_VEL
LIN {X 0,Y 418.318,Z 298.38,A -85,B 0,C 180,E1 -10063.405,E2 -10063.405} C_VEL
LIN {X 0,Y 418.347,Z 298.368,A -85,B 0,C 180,E1 -10066.999,E2 -10066.999} C_VEL
LIN {X 0,Y 418.341,Z 298.364,A -85,B 0,C 180,E1 -10070.329,E2 -10070.329} C_VEL
LIN {X 0,Y 418.514,Z 298.351,A -85,B 0,C 180,E1 -10072.279,E2 -10072.279} C_VEL
LIN {X 0,Y 418.509,Z 298.349,A -85,B 0,C 180,E1 -10074.217,E2 -10074.217} C_VEL
LIN {X 0,Y 418.542,Z 298.35,A -85,B 0,C 180,E1 -10078.075,E2 -10078.075} C_VEL
LIN {X 0,Y 418.671,Z 298.327,A -85,B 0,C 180,E1 -10080,E2 -10080} C_VEL
LIN {X 0,Y 418.501,Z 298.349,A -85,B 0,C 180,E1 -10082.888,E2 -10082.888} C_VEL
LIN {X 0,Y 418.491,Z 298.349,A -85,B 0,C 180,E1 -10086.751,E2 -10086.751} C_VEL
LIN {X 0,Y 418.4,Z 298.364,A -85,B 0,C 180,E1 -10088.695,E2 -10088.695} C_VEL
LIN {X 0,Y 418.356,Z 298.372,A -85,B 0,C 180,E1 -10092.614,E2 -10092.614} C_VEL
LIN {X 0,Y 418.302,Z 298.371,A -85,B 0,C 180,E1 -10095.594,E2 -10095.594} C_VEL
